  MoveL 5376 to (-21.97, 164.98, 78.65) mm, rotated rx 180 ry 0 rz 180 deg; joints [-137.804, 64.103, -73.918, 137.384, 82.745, 6.628]
  Call Extruder(394.83845)
  MoveL 5377 to (-22.56, 164.93, 78.65) mm, rotated rx -180 ry 0 rz 180 deg; joints [-137.905, 64.127, -73.891, 137.489, 82.771, 6.581]
  MoveL 5378 to (-22.56, 164.93, 78.65) mm, rotated rx -180 ry 0 rz 180 deg; joints [-137.905, 64.127, -73.891, 137.489, 82.771, 6.581]
  Call Extruder(395.13381)
  MoveL 5379 to (-23.15, 164.89, 78.65) mm, rotated rx 180 ry 0 rz -180 deg; joints [-138.004, 64.152, -73.865, 137.593, 82.796, 6.534]
  MoveL 5380 to (-23.15, 164.89, 78.65) mm, rotated rx 180 ry 0 rz -180 deg; joints [-138.004, 64.152, -73.865, 137.593, 82.796, 6.534]
  Call Extruder(395.38003)
  MoveL 5381 to (-23.64, 164.84, 78.65) mm, rotated rx 180 ry 0 rz 180 deg; joints [-138.088, 64.171, -73.843, 137.68, 82.818, 6.495]
  MoveL 5382 to (-23.64, 164.84, 78.65) mm, rotated rx 180 ry 0 rz 180 deg; joints [-138.088, 64.171, -73.843, 137.68, 82.818, 6.495]
  Call Extruder(395.57673)
  MoveL 5383 to (-24.03, 164.79, 78.65) mm, rotated rx 180 ry 0 rz 180 deg; joints [-138.156, 64.187, -73.827, 137.751, 82.834, 6.465]
  MoveL 5384 to (-24.03, 164.79, 78.65) mm, rotated rx 180 ry 0 rz 180 deg; joints [-138.156, 64.187, -73.827, 137.751, 82.834, 6.465]
  Call Extruder(395.77431)
  MoveL 5385 to (-24.42, 164.75, 78.65) mm, rotated rx 180 ry 0 rz 180 deg; joints [-138.224, 64.202, -73.81, 137.822, 82.85, 6.434]
  MoveL 5386 to (-24.42, 164.75, 78.65) mm, rotated rx 180 ry 0 rz 180 deg; joints [-138.224, 64.202, -73.81, 137.822, 82.85, 6.434]
  Call Extruder(395.97275)
  MoveL 5387 to (-24.8, 164.7, 78.65) mm, rotated rx -180 ry 0 rz -180 deg; joints [-138.292, 64.217, -73.793, 137.892, 82.866, 6.404]
  MoveL 5388 to (-24.8, 164.7, 78.65) mm, rotated rx -180 ry 0 rz -180 deg; joints [-138.292, 64.217, -73.793, 137.892, 82.866, 6.404]
  Call Extruder(396.17206)
  MoveL 5389 to (-25.19, 164.66, 78.65) mm, rotated rx 180 ry 0 rz 180 deg; joints [-138.359, 64.233, -73.776, 137.962, 82.883, 6.374]
  MoveL 5390 to (-25.19, 164.66, 78.65) mm, rotated rx 180 ry 0 rz 180 deg; joints [-138.359, 64.233, -73.776, 137.962, 82.883, 6.374]
  Call Extruder(396.33089)
  MoveL 5391 to (-25.5, 164.61, 78.65) mm, rotated rx -180 ry 0 rz 180 deg; joints [-138.415, 64.244, -73.763, 138.02, 82.895, 6.351]
  MoveL 5392 to (-25.5, 164.61, 78.65) mm, rotated rx -180 ry 0 rz 180 deg; joints [-138.415, 64.244, -73.763, 138.02, 82.895, 6.351]
  Call Extruder(396.49045)
  MoveL 5393 to (-25.8, 164.56, 78.65) mm, rotated rx -180 ry 0 rz 180 deg; joints [-138.47, 64.256, -73.75, 138.077, 82.907, 6.327]
  MoveL 5394 to (-25.8, 164.56, 78.65) mm, rotated rx -180 ry 0 rz 180 deg; joints [-138.47, 64.256, -73.75, 138.077, 82.907, 6.327]
  Call Extruder(396.65073)
  MoveL 5395 to (-26.11, 164.51, 78.65) mm, rotated rx 180 ry 0 rz 180 deg; joints [-138.525, 64.267, -73.737, 138.134, 82.919, 6.304]
  MoveL 5396 to (-26.11, 164.51, 78.65) mm, rotated rx 180 ry 0 rz 180 deg; joints [-138.525, 64.267, -73.737, 138.134, 82.919, 6.304]
  Call Extruder(396.81175)
  MoveL 5397 to (-26.41, 164.46, 78.65) mm, rotated rx 180 ry 0 rz 180 deg; joints [-138.58, 64.279, -73.724, 138.192, 82.931, 6.281]
  MoveL 5398 to (-26.41, 164.46, 78.65) mm, rotated rx 180 ry 0 rz 180 deg; joints [-138.58, 64.279, -73.724, 138.192, 82.931, 6.281]
  Call Extruder(396.97349)
  MoveL 5399 to (-26.72, 164.41, 78.65) mm, rotated rx 180 ry 0 rz 180 deg; joints [-138.635, 64.291, -73.711, 138.249, 82.944, 6.257]
  MoveL 5400 to (-26.72, 164.41, 78.65) mm, rotated rx 180 ry 0 rz 180 deg; joints [-138.635, 64.291, -73.711, 138.249, 82.944, 6.257]
  Call Extruder(397.13596)
  MoveL 5401 to (-27.03, 164.37, 78.65) mm, rotated rx 180 ry 0 rz 180 deg; joints [-138.69, 64.302, -73.698, 138.306, 82.956, 6.234]
  MoveL 5402 to (-27.03, 164.37, 78.65) mm, rotated rx 180 ry 0 rz 180 deg; joints [-138.69, 64.302, -73.698, 138.306, 82.956, 6.234]
  Call Extruder(397.26988)
  MoveL 5403 to (-27.27, 164.32, 78.65) mm, rotated rx -180 ry 0 rz 180 deg; joints [-138.736, 64.311, -73.688, 138.354, 82.965, 6.216]
  MoveL 5404 to (-27.27, 164.32, 78.65) mm, rotated rx -180 ry 0 rz 180 deg; joints [-138.736, 64.311, -73.688, 138.354, 82.965, 6.216]
  Call Extruder(397.40442)
  MoveL 5405 to (-27.52, 164.27, 78.65) mm, rotated rx 180 ry 0 rz 180 deg; joints [-138.783, 64.32, -73.678, 138.402, 82.975, 6.197]
  MoveL 5406 to (-27.52, 164.27, 78.65) mm, rotated rx 180 ry 0 rz 180 deg; joints [-138.783, 64.32, -73.678, 138.402, 82.975, 6.197]
  Call Extruder(397.53957)
  MoveL 5407 to (-27.77, 164.22, 78.65) mm, rotated rx 180 ry 0 rz 180 deg; joints [-138.829, 64.329, -73.668, 138.45, 82.984, 6.178]
  MoveL 5408 to (-27.77, 164.22, 78.65) mm, rotated rx 180 ry 0 rz 180 deg; joints [-138.829, 64.329, -73.668, 138.45, 82.984, 6.178]
  Call Extruder(397.67532)
  MoveL 5409 to (-28.02, 164.17, 78.65) mm, rotated rx -180 ry 0 rz 180 deg; joints [-138.875, 64.338, -73.657, 138.497, 82.994, 6.16]
  MoveL 5410 to (-28.02, 164.17, 78.65) mm, rotated rx -180 ry 0 rz 180 deg; joints [-138.875, 64.338, -73.657, 138.497, 82.994, 6.16]
  Call Extruder(397.81169)
  MoveL 5411 to (-28.27, 164.12, 78.65) mm, rotated rx -180 ry 0 rz -180 deg; joints [-138.921, 64.348, -73.647, 138.545, 83.003, 6.141]
  MoveL 5412 to (-28.27, 164.12, 78.65) mm, rotated rx -180 ry 0 rz -180 deg; joints [-138.921, 64.348, -73.647, 138.545, 83.003, 6.141]
  Call Extruder(397.89656)
  MoveL 5413 to (-28.42, 164.09, 78.65) mm, rotated rx -180 ry 0 rz 180 deg; joints [-138.95, 64.353, -73.641, 138.575, 83.009, 6.13]
  Set speed (130.0 mm/s)
  MoveL 5414 to (-31.76, 163.31, 78.65) mm, rotated rx -180 ry 0 rz 180 deg; joints [-139.581, 64.47, -73.506, 139.228, 83.133, 5.887]
  MoveL 5415 to (-31.76, 163.31, 88.06) mm, rotated rx -180 ry 0 rz -180 deg; joints [-139.581, 65.843, -75.425, 139.183, 82.719, 6.247]
  Call Extruder(395.89656)
  Set speed (40.0 mm/s)
  MoveL 5416 to (-31.76, 163.31, 88.06) mm, rotated rx -180 ry 0 rz -180 deg; joints [-139.581, 65.843, -75.425, 139.183, 82.719, 6.247]
  Call Extruder(0.00000)
  Set speed (130.0 mm/s)
  MoveL 5417 to (-31.64, 163.21, 88.06) mm, rotated rx -180 ry 0 rz 180 deg; joints [-139.581, 65.833, -75.436, 139.181, 82.704, 6.26]
  Call Extruder(2.00000)
  Set speed (40.0 mm/s)
  MoveL 5418 to (-31.64, 163.21, 88.06) mm, rotated rx -180 ry 0 rz 180 deg; joints [-139.581, 65.833, -75.436, 139.181, 82.704, 6.26]
  Set speed (30.0 mm/s)
  MoveL 5419 to (-31.64, 163.21, 88.06) mm, rotated rx -180 ry 0 rz 180 deg; joints [-139.581, 65.833, -75.436, 139.181, 82.704, 6.26]
  Call Extruder(2.18198)
  MoveL 5420 to (-31.93, 163.09, 88.06) mm, rotated rx -180 ry 0 rz 180 deg; joints [-139.645, 65.842, -75.426, 139.247, 82.711, 6.24]
  MoveL 5421 to (-31.93, 163.09, 88.06) mm, rotated rx -180 ry 0 rz 180 deg; joints [-139.645, 65.842, -75.426, 139.247, 82.711, 6.24]
  Call Extruder(2.36471)
  MoveL 5422 to (-32.22, 162.96, 88.06) mm, rotated rx -180 ry 0 rz 180 deg; joints [-139.709, 65.851, -75.416, 139.313, 82.718, 6.219]
  MoveL 5423 to (-32.22, 162.96, 88.06) mm, rotated rx -180 ry 0 rz 180 deg; joints [-139.709, 65.851, -75.416, 139.313, 82.718, 6.219]
  Call Extruder(2.53513)
  MoveL 5424 to (-32.49, 162.85, 88.06) mm, rotated rx -180 ry 0 rz -180 deg; joints [-139.768, 65.858, -75.407, 139.374, 82.724, 6.201]
  MoveL 5425 to (-32.49, 162.85, 88.06) mm, rotated rx -180 ry 0 rz -180 deg; joints [-139.768, 65.858, -75.407, 139.374, 82.724, 6.201]
  Call Extruder(2.69310)
  MoveL 5426 to (-32.74, 162.74, 88.06) mm, rotated rx -180 ry 0 rz 180 deg; joints [-139.823, 65.866, -75.399, 139.43, 82.73, 6.184]
  MoveL 5427 to (-32.74, 162.74, 88.06) mm, rotated rx -180 ry 0 rz 180 deg; joints [-139.823, 65.866, -75.399, 139.43, 82.73, 6.184]
  Call Extruder(2.85168)
  MoveL 5428 to (-32.99, 162.64, 88.06) mm, rotated rx -180 ry 0 rz 180 deg; joints [-139.878, 65.873, -75.391, 139.487, 82.736, 6.167]
  MoveL 5429 to (-32.99, 162.64, 88.06) mm, rotated rx -180 ry 0 rz 180 deg; joints [-139.878, 65.873, -75.391, 139.487, 82.736, 6.167]
  Call Extruder(3.05785)
  MoveL 5430 to (-33.29, 162.46, 88.06) mm, rotated rx -180 ry 0 rz 180 deg; joints [-139.953, 65.88, -75.383, 139.563, 82.739, 6.147]
  MoveL 5431 to (-33.29, 162.46, 88.06) mm, rotated rx -180 ry 0 rz 180 deg; joints [-139.953, 65.88, -75.383, 139.563, 82.739, 6.147]
  Call Extruder(3.26479)
  MoveL 5432 to (-33.6, 162.29, 88.06) mm, rotated rx -180 ry 0 rz 180 deg; joints [-140.028, 65.887, -75.375, 139.639, 82.743, 6.128]
  MoveL 5433 to (-33.6, 162.29, 88.06) mm, rotated rx -180 ry 0 rz 180 deg; joints [-140.028, 65.887, -75.375, 139.639, 82.743, 6.128]
  Call Extruder(3.47251)
  MoveL 5434 to (-33.9, 162.11, 88.06) mm, rotated rx 180 ry 0 rz -180 deg; joints [-140.103, 65.894, -75.367, 139.715, 82.746, 6.109]
  MoveL 5435 to (-33.9, 162.11, 88.06) mm, rotated rx 180 ry 0 rz -180 deg; joints [-140.103, 65.894, -75.367, 139.715, 82.746, 6.109]
  Call Extruder(3.68102)
  MoveL 5436 to (-34.21, 161.93, 88.06) mm, rotated rx -180 ry 0 rz 180 deg; joints [-140.178, 65.901, -75.359, 139.791, 82.75, 6.089]
  MoveL 5437 to (-34.21, 161.93, 88.06) mm, rotated rx -180 ry 0 rz 180 deg; joints [-140.178, 65.901, -75.359, 139.791, 82.75, 6.089]
  Call Extruder(3.86055)
  MoveL 5438 to (-34.45, 161.76, 88.06) mm, rotated rx -180 ry 0 rz 180 deg; joints [-140.244, 65.905, -75.354, 139.859, 82.75, 6.075]
  MoveL 5439 to (-34.45, 161.76, 88.06) mm, rotated rx -180 ry 0 rz 180 deg; joints [-140.244, 65.905, -75.354, 139.859, 82.75, 6.075]
  Call Extruder(4.19399)
  MoveL 5440 to (-34.9, 161.43, 88.06) mm, rotated rx 180 ry 0 rz 180 deg; joints [-140.366, 65.914, -75.344, 139.983, 82.75, 6.048]
  MoveL 5441 to (-34.9, 161.43, 88.06) mm, rotated rx 180 ry 0 rz 180 deg; joints [-140.366, 65.914, -75.344, 139.983, 82.75, 6.048]
  Call Extruder(4.52861)
  MoveL 5442 to (-35.35, 161.1, 88.06) mm, rotated rx -180 ry 0 rz -180 deg; joints [-140.489, 65.922, -75.335, 140.107, 82.751, 6.021]
  Call Extruder(5.35652)
  MoveL 5443 to (-36.39, 160.19, 88.06) mm, rotated rx -180 ry 0 rz -180 deg; joints [-140.797, 65.935, -75.32, 140.418, 82.741, 5.964]
  Call Extruder(6.18445)
  MoveL 5444 to (-37.3, 159.15, 88.06) mm, rotated rx 180 ry 0 rz 180 deg; joints [-141.109, 65.938, -75.316, 140.731, 82.714, 5.92]
  Call Extruder(6.35176)
  MoveL 5445 to (-37.47, 158.93, 88.06) mm, rotated rx 180 ry 0 rz 180 deg; joints [-141.172, 65.937, -75.317, 140.795, 82.706, 5.913]
  MoveL 5446 to (-37.47, 158.93, 88.06) mm, rotated rx 180 ry 0 rz 180 deg; joints [-141.172, 65.937, -75.317, 140.795, 82.706, 5.913]
  Call Extruder(6.68519)
  MoveL 5447 to (-37.79, 158.48, 88.06) mm, rotated rx -180 ry 0 rz 180 deg; joints [-141.298, 65.936, -75.319, 140.921, 82.69, 5.899]
  MoveL 5448 to (-37.79, 158.48, 88.06) mm, rotated rx -180 ry 0 rz 180 deg; joints [-141.298, 65.936, -75.319, 140.921, 82.69, 5.899]
  Call Extruder(7.01743)
  MoveL 5449 to (-38.12, 158.03, 88.06) mm, rotated rx -180 ry 0 rz 180 deg; joints [-141.424, 65.934, -75.321, 141.047, 82.675, 5.885]
  MoveL 5450 to (-38.12, 158.03, 88.06) mm, rotated rx -180 ry 0 rz 180 deg; joints [-141.424, 65.934, -75.321, 141.047, 82.675, 5.885]
  Call Extruder(7.13510)
  MoveL 5451 to (-38.22, 157.85, 88.06) mm, rotated rx 180 ry 0 rz -180 deg; joints [-141.468, 65.932, -75.323, 141.091, 82.667, 5.882]
  MoveL 5452 to (-38.22, 157.85, 88.06) mm, rotated rx 180 ry 0 rz -180 deg; joints [-141.468, 65.932, -75.323, 141.091, 82.667, 5.882]
  Call Extruder(7.34283)
  MoveL 5453 to (-38.4, 157.55, 88.06) mm, rotated rx -180 ry 0 rz 180 deg; joints [-141.547, 65.929, -75.326, 141.169, 82.654, 5.876]
  MoveL 5454 to (-38.4, 157.55, 88.06) mm, rotated rx -180 ry 0 rz 180 deg; joints [-141.547, 65.929, -75.326, 141.169, 82.654, 5.876]
  Call Extruder(7.54978)
  MoveL 5455 to (-38.57, 157.25, 88.06) mm, rotated rx -180 ry 0 rz 180 deg; joints [-141.625, 65.926, -75.329, 141.247, 82.641, 5.87]
  MoveL 5456 to (-38.57, 157.25, 88.06) mm, rotated rx -180 ry 0 rz 180 deg; joints [-141.625, 65.926, -75.329, 141.247, 82.641, 5.87]
  Call Extruder(7.75595)
  MoveL 5457 to (-38.75, 156.94, 88.06) mm, rotated rx 180 ry 0 rz 180 deg; joints [-141.704, 65.923, -75.333, 141.326, 82.628, 5.864]
  MoveL 5458 to (-38.75, 156.94, 88.06) mm, rotated rx 180 ry 0 rz 180 deg; joints [-141.704, 65.923, -75.333, 141.326, 82.628, 5.864]
  Call Extruder(7.93763)
  MoveL 5459 to (-38.89, 156.66, 88.06) mm, rotated rx -180 ry 0 rz 180 deg; joints [-141.773, 65.92, -75.337, 141.394, 82.615, 5.86]
  MoveL 5460 to (-38.89, 156.66, 88.06) mm, rotated rx -180 ry 0 rz 180 deg; joints [-141.773, 65.92, -75.337, 141.394, 82.615, 5.86]
  Call Extruder(8.09561)
  MoveL 5461 to (-39, 156.42, 88.06) mm, rotated rx -180 ry 0 rz 180 deg; joints [-141.832, 65.916, -75.342, 141.453, 82.602, 5.858]
  MoveL 5462 to (-39, 156.42, 88.06) mm, rotated rx -180 ry 0 rz 180 deg; joints [-141.832, 65.916, -75.342, 141.453, 82.602, 5.858]
  Call Extruder(8.25300)
  MoveL 5463 to (-39.11, 156.17, 88.06) mm, rotated rx -180 ry 0 rz 180 deg; joints [-141.891, 65.912, -75.346, 141.512, 82.589, 5.855]
  MoveL 5464 to (-39.11, 156.17, 88.06) mm, rotated rx -180 ry 0 rz 180 deg; joints [-141.891, 65.912, -75.346, 141.512, 82.589, 5.855]
  Call Extruder(8.43571)
  MoveL 5465 to (-39.23, 155.87, 88.06) mm, rotated rx -180 ry 0 rz -180 deg; joints [-141.96, 65.907, -75.352, 141.58, 82.574, 5.853]
  MoveL 5466 to (-39.23, 155.87, 88.06) mm, rotated rx -180 ry 0 rz -180 deg; joints [-141.96, 65.907, -75.352, 141.58, 82.574, 5.853]
  Call Extruder(8.61768)
  MoveL 5467 to (-39.35, 155.58, 88.06) mm, rotated rx 180 ry 0 rz 180 deg; joints [-142.029, 65.902, -75.358, 141.648, 82.558, 5.851]
  MoveL 5468 to (-39.35, 155.58, 88.06) mm, rotated rx 180 ry 0 rz 180 deg; joints [-142.029, 65.902, -75.358, 141.648, 82.558, 5.851]
  Call Extruder(8.76501)
  MoveL 5469 to (-39.44, 155.34, 88.06) mm, rotated rx 180 ry 0 rz -180 deg; joints [-142.085, 65.897, -75.363, 141.703, 82.545, 5.85]
  MoveL 5470 to (-39.44, 155.34, 88.06) mm, rotated rx 180 ry 0 rz -180 deg; joints [-142.085, 65.897, -75.363, 141.703, 82.545, 5.85]
  Call Extruder(8.87824)
  MoveL 5471 to (-39.5, 155.15, 88.06) mm, rotated rx -180 ry 0 rz -180 deg; joints [-142.127, 65.893, -75.367, 141.745, 82.534, 5.85]
  MoveL 5472 to (-39.5, 155.15, 88.06) mm, rotated rx -180 ry 0 rz -180 deg; joints [-142.127, 65.893, -75.367, 141.745, 82.534, 5.85]
  Call Extruder(8.99103)
  MoveL 5473 to (-39.56, 154.97, 88.06) mm, rotated rx 180 ry 0 rz 180 deg; joints [-142.169, 65.889, -75.372, 141.787, 82.523, 5.849]
  MoveL 5474 to (-39.56, 154.97, 88.06) mm, rotated rx 180 ry 0 rz 180 deg; joints [-142.169, 65.889, -75.372, 141.787, 82.523, 5.849]
  Call Extruder(9.10338)
  MoveL 5475 to (-39.62, 154.78, 88.06) mm, rotated rx -180 ry 0 rz 180 deg; joints [-142.212, 65.885, -75.377, 141.829, 82.512, 5.849]
  MoveL 5476 to (-39.62, 154.78, 88.06) mm, rotated rx -180 ry 0 rz 180 deg; joints [-142.212, 65.885, -75.377, 141.829, 82.512, 5.849]
  Call Extruder(9.21528)
  MoveL 5477 to (-39.68, 154.59, 88.06) mm, rotated rx -180 ry 0 rz -180 deg; joints [-142.254, 65.881, -75.381, 141.87, 82.501, 5.849]
  MoveL 5478 to (-39.68, 154.59, 88.06) mm, rotated rx -180 ry 0 rz -180 deg; joints [-142.254, 65.881, -75.381, 141.87, 82.501, 5.849]
  Call Extruder(9.33668)
  MoveL 5479 to (-39.75, 154.38, 88.06) mm, rotated rx -180 ry 0 rz 180 deg; joints [-142.3, 65.877, -75.386, 141.916, 82.489, 5.849]
  MoveL 5480 to (-39.75, 154.38, 88.06) mm, rotated rx -180 ry 0 rz 180 deg; joints [-142.3, 65.877, -75.386, 141.916, 82.489, 5.849]
  Call Extruder(9.46747)
  MoveL 5481 to (-39.82, 154.16, 88.06) mm, rotated rx 180 ry 0 rz 180 deg; joints [-142.35, 65.872, -75.392, 141.965, 82.476, 5.849]
  MoveL 5482 to (-39.82, 154.16, 88.06) mm, rotated rx 180 ry 0 rz 180 deg; joints [-142.35, 65.872, -75.392, 141.965, 82.476, 5.849]
  Call Extruder(9.59770)
  MoveL 5483 to (-39.88, 153.94, 88.06) mm, rotated rx 180 ry 0 rz -180 deg; joints [-142.399, 65.867, -75.397, 142.013, 82.463, 5.849]
  MoveL 5484 to (-39.88, 153.94, 88.06) mm, rotated rx 180 ry 0 rz -180 deg; joints [-142.399, 65.867, -75.397, 142.013, 82.463, 5.849]
  Call Extruder(9.72737)
  MoveL 5485 to (-39.95, 153.71, 88.06) mm, rotated rx -180 ry 0 rz -180 deg; joints [-142.449, 65.862, -75.403, 142.062, 82.449, 5.849]
  MoveL 5486 to (-39.95, 153.71, 88.06) mm, rotated rx -180 ry 0 rz -180 deg; joints [-142.449, 65.862, -75.403, 142.062, 82.449, 5.849]
  Call Extruder(9.85647)
  MoveL 5487 to (-40.02, 153.49, 88.06) mm, rotated rx -180 ry 0 rz 180 deg; joints [-142.498, 65.857, -75.408, 142.111, 82.436, 5.849]
  MoveL 5488 to (-40.02, 153.49, 88.06) mm, rotated rx -180 ry 0 rz 180 deg; joints [-142.498, 65.857, -75.408, 142.111, 82.436, 5.849]
  Call Extruder(9.97156)
  MoveL 5489 to (-40.06, 153.28, 88.06) mm, rotated rx -180 ry 0 rz 180 deg; joints [-142.541, 65.852, -75.414, 142.154, 82.423, 5.85]
  MoveL 5490 to (-40.06, 153.28, 88.06) mm, rotated rx -180 ry 0 rz 180 deg; joints [-142.541, 65.852, -75.414, 142.154, 82.423, 5.85]
  Call Extruder(10.08619)
  MoveL 5491 to (-40.11, 153.08, 88.06) mm, rotated rx 180 ry 0 rz 180 deg; joints [-142.584, 65.847, -75.42, 142.196, 82.41, 5.851]
  MoveL 5492 to (-40.11, 153.08, 88.06) mm, rotated rx 180 ry 0 rz 180 deg; joints [-142.584, 65.847, -75.42, 142.196, 82.41, 5.851]
  Call Extruder(10.20038)
  MoveL 5493 to (-40.15, 152.88, 88.06) mm, rotated rx 180 ry 0 rz 180 deg; joints [-142.627, 65.842, -75.426, 142.238, 82.396, 5.852]
  MoveL 5494 to (-40.15, 152.88, 88.06) mm, rotated rx 180 ry 0 rz 180 deg; joints [-142.627, 65.842, -75.426, 142.238, 82.396, 5.852]
  Call Extruder(10.31411)
  MoveL 5495 to (-40.2, 152.67, 88.06) mm, rotated rx -180 ry 0 rz 180 deg; joints [-142.671, 65.836, -75.432, 142.281, 82.383, 5.853]
  MoveL 5496 to (-40.2, 152.67, 88.06) mm, rotated rx -180 ry 0 rz 180 deg; joints [-142.671, 65.836, -75.432, 142.281, 82.383, 5.853]
  Call Extruder(10.43953)
  MoveL 5497 to (-40.24, 152.44, 88.06) mm, rotated rx 180 ry 0 rz 180 deg; joints [-142.718, 65.831, -75.439, 142.327, 82.368, 5.855]
  MoveL 5498 to (-40.24, 152.44, 88.06) mm, rotated rx 180 ry 0 rz 180 deg; joints [-142.718, 65.831, -75.439, 142.327, 82.368, 5.855]
  Call Extruder(10.57651)
  MoveL 5499 to (-40.29, 152.2, 88.06) mm, rotated rx 180 ry 0 rz 180 deg; joints [-142.77, 65.824, -75.446, 142.378, 82.352, 5.856]
  MoveL 5500 to (-40.29, 152.2, 88.06) mm, rotated rx 180 ry 0 rz 180 deg; joints [-142.77, 65.824, -75.446, 142.378, 82.352, 5.856]
  Call Extruder(10.71287)
  MoveL 5501 to (-40.34, 151.95, 88.06) mm, rotated rx -180 ry 0 rz 180 deg; joints [-142.822, 65.817, -75.454, 142.429, 82.335, 5.858]
  MoveL 5502 to (-40.34, 151.95, 88.06) mm, rotated rx -180 ry 0 rz 180 deg; joints [-142.822, 65.817, -75.454, 142.429, 82.335, 5.858]
  Call Extruder(10.84863)
  MoveL 5503 to (-40.39, 151.7, 88.06) mm, rotated rx 180 ry 0 rz 180 deg; joints [-142.874, 65.811, -75.461, 142.481, 82.319, 5.86]
  MoveL 5504 to (-40.39, 151.7, 88.06) mm, rotated rx 180 ry 0 rz 180 deg; joints [-142.874, 65.811, -75.461, 142.481, 82.319, 5.86]
  Call Extruder(10.98377)
  MoveL 5505 to (-40.44, 151.45, 88.06) mm, rotated rx -180 ry 0 rz 180 deg; joints [-142.926, 65.804, -75.468, 142.532, 82.303, 5.861]
  MoveL 5506 to (-40.44, 151.45, 88.06) mm, rotated rx -180 ry 0 rz 180 deg; joints [-142.926, 65.804, -75.468, 142.532, 82.303, 5.861]
  Call Extruder(11.11831)
  MoveL 5507 to (-40.49, 151.2, 88.06) mm, rotated rx 180 ry 0 rz 180 deg; joints [-142.978, 65.798, -75.476, 142.583, 82.286, 5.863]
  MoveL 5508 to (-40.49, 151.2, 88.06) mm, rotated rx 180 ry 0 rz 180 deg; joints [-142.978, 65.798, -75.476, 142.583, 82.286, 5.863]
  Call Extruder(11.25223)
  MoveL 5509 to (-40.54, 150.95, 88.06) mm, rotated rx 180 ry 0 rz 180 deg; joints [-143.031, 65.791, -75.483, 142.634, 82.27, 5.864]
  MoveL 5510 to (-40.54, 150.95, 88.06) mm, rotated rx 180 ry 0 rz 180 deg; joints [-143.031, 65.791, -75.483, 142.634, 82.27, 5.864]
  Call Extruder(11.40009)
  MoveL 5511 to (-40.59, 150.67, 88.06) mm, rotated rx 180 ry 0 rz 180 deg; joints [-143.088, 65.784, -75.492, 142.69, 82.251, 5.866]
  MoveL 5512 to (-40.59, 150.67, 88.06) mm, rotated rx 180 ry 0 rz 180 deg; joints [-143.088, 65.784, -75.492, 142.69, 82.251, 5.866]
  Call Extruder(11.56181)
  MoveL 5513 to (-40.64, 150.37, 88.06) mm, rotated rx -180 ry 0 rz 180 deg; joints [-143.15, 65.775, -75.501, 142.752, 82.23, 5.869]
  MoveL 5514 to (-40.64, 150.37, 88.06) mm, rotated rx -180 ry 0 rz 180 deg; joints [-143.15, 65.775, -75.501, 142.752, 82.23, 5.869]
  Call Extruder(11.72281)
  MoveL 5515 to (-40.69, 150.06, 88.06) mm, rotated rx -180 ry 0 rz 180 deg; joints [-143.213, 65.766, -75.511, 142.813, 82.209, 5.872]
  MoveL 5516 to (-40.69, 150.06, 88.06) mm, rotated rx -180 ry 0 rz 180 deg; joints [-143.213, 65.766, -75.511, 142.813, 82.209, 5.872]
  Call Extruder(11.88308)
  MoveL 5517 to (-40.74, 149.76, 88.06) mm, rotated rx -180 ry 0 rz 180 deg; joints [-143.276, 65.758, -75.52, 142.874, 82.189, 5.874]
  MoveL 5518 to (-40.74, 149.76, 88.06) mm, rotated rx -180 ry 0 rz 180 deg; joints [-143.276, 65.758, -75.52, 142.874, 82.189, 5.874]
  Call Extruder(12.04262)
  MoveL 5519 to (-40.78, 149.45, 88.06) mm, rotated rx -180 ry 0 rz -180 deg; joints [-143.338, 65.749, -75.53, 142.936, 82.168, 5.877]
  MoveL 5520 to (-40.78, 149.45, 88.06) mm, rotated rx -180 ry 0 rz -180 deg; joints [-143.338, 65.749, -75.53, 142.936, 82.168, 5.877]
  Call Extruder(12.20144)
  MoveL 5521 to (-40.83, 149.14, 88.06) mm, rotated rx 180 ry 0 rz 180 deg; joints [-143.401, 65.741, -75.54, 142.997, 82.147, 5.879]
  MoveL 5522 to (-40.83, 149.14, 88.06) mm, rotated rx 180 ry 0 rz 180 deg; joints [-143.401, 65.741, -75.54, 142.997, 82.147, 5.879]
  Call Extruder(12.38010)
  MoveL 5523 to (-40.88, 148.8, 88.06) mm, rotated rx -180 ry 0 rz 180 deg; joints [-143.471, 65.731, -75.551, 143.066, 82.123, 5.882]
  MoveL 5524 to (-40.88, 148.8, 88.06) mm, rotated rx -180 ry 0 rz 180 deg; joints [-143.471, 65.731, -75.551, 143.066, 82.123, 5.882]
  Call Extruder(12.57854)
  MoveL 5525 to (-40.92, 148.41, 88.06) mm, rotated rx -180 ry 0 rz 180 deg; joints [-143.549, 65.719, -75.564, 143.142, 82.095, 5.886]
  MoveL 5526 to (-40.92, 148.41, 88.06) mm, rotated rx -180 ry 0 rz 180 deg; joints [-143.549, 65.719, -75.564, 143.142, 82.095, 5.886]
  Call Extruder(12.77611)
  MoveL 5527 to (-40.97, 148.02, 88.06) mm, rotated rx -180 ry 0 rz -180 deg; joints [-143.627, 65.708, -75.576, 143.218, 82.068, 5.89]
  MoveL 5528 to (-40.97, 148.02, 88.06) mm, rotated rx -180 ry 0 rz -180 deg; joints [-143.627, 65.708, -75.576, 143.218, 82.068, 5.89]
  Call Extruder(12.97282)
  MoveL 5529 to (-41.02, 147.63, 88.06) mm, rotated rx -180 ry 0 rz -180 deg; joints [-143.705, 65.696, -75.589, 143.295, 82.04, 5.894]
  MoveL 5530 to (-41.02, 147.63, 88.06) mm, rotated rx -180 ry 0 rz -180 deg; joints [-143.705, 65.696, -75.589, 143.295, 82.04, 5.894]
  Call Extruder(13.16866)
  MoveL 5531 to (-41.06, 147.25, 88.06) mm, rotated rx -180 ry 0 rz 180 deg; joints [-143.783, 65.684, -75.602, 143.371, 82.013, 5.898]
  MoveL 5532 to (-41.06, 147.25, 88.06) mm, rotated rx -180 ry 0 rz 180 deg; joints [-143.783, 65.684, -75.602, 143.371, 82.013, 5.898]
  Call Extruder(13.46406)
  MoveL 5533 to (-41.11, 146.66, 88.06) mm, rotated rx -180 ry 0 rz -180 deg; joints [-143.899, 65.666, -75.622, 143.484, 81.97, 5.905]
  MoveL 5534 to (-41.11, 146.66, 88.06) mm, rotated rx -180 ry 0 rz -180 deg; joints [-143.899, 65.666, -75.622, 143.484, 81.97, 5.905]
  Call Extruder(13.75812)
  MoveL 5535 to (-41.16, 146.07, 88.06) mm, rotated rx -180 ry 0 rz 180 deg; joints [-144.015, 65.647, -75.643, 143.597, 81.926, 5.912]
  MoveL 5536 to (-41.16, 146.07, 88.06) mm, rotated rx -180 ry 0 rz 180 deg; joints [-144.015, 65.647, -75.643, 143.597, 81.926, 5.912]
  Call Extruder(14.05085)
  MoveL 5537 to (-41.2, 145.48, 88.06) mm, rotated rx -180 ry 0 rz 180 deg; joints [-144.131, 65.629, -75.663, 143.711, 81.883, 5.919]
  MoveL 5538 to (-41.2, 145.48, 88.06) mm, rotated rx -180 ry 0 rz 180 deg; joints [-144.131, 65.629, -75.663, 143.711, 81.883, 5.919]
  Call Extruder(14.62431)
  MoveL 5539 to (-41.25, 144.32, 88.06) mm, rotated rx -180 ry 0 rz -180 deg; joints [-144.355, 65.59, -75.705, 143.929, 81.795, 5.935]
  MoveL 5540 to (-41.25, 144.32, 88.06) mm, rotated rx -180 ry 0 rz -180 deg; joints [-144.355, 65.59, -75.705, 143.929, 81.795, 5.935]
  Call Extruder(15.33827)
  MoveL 5541 to (-41.29, 142.86, 88.06) mm, rotated rx 180 ry 0 rz 180 deg; joints [-144.635, 65.541, -75.758, 144.202, 81.683, 5.955]
  Call Extruder(57.40309)
  MoveL 5542 to (-41.29, 57.14, 88.06) mm, rotated rx -180 ry 0 rz -180 deg; joints [-164.153, 63.039, -77.935, 163.631, 75.682, 4.155]
  Call Extruder(57.83165)
  MoveL 5543 to (-41.27, 56.26, 88.06) mm, rotated rx -180 ry 0 rz 180 deg; joints [-164.382, 63.02, -77.948, 163.864, 75.636, 4.105]
  MoveL 5544 to (-41.27, 56.26, 88.06) mm, rotated rx -180 ry 0 rz 180 deg; joints [-164.382, 63.02, -77.948, 163.864, 75.636, 4.105]
  Call Extruder(58.40510)
  MoveL 5545 to (-41.23, 55.1, 88.06) mm, rotated rx -180 ry 0 rz 180 deg; joints [-164.686, 62.995, -77.965, 164.174, 75.572, 4.04]
  MoveL 5546 to (-41.23, 55.1, 88.06) mm, rotated rx -180 ry 0 rz 180 deg; joints [-164.686, 62.995, -77.965, 164.174, 75.572, 4.04]
  Call Extruder(58.83942)
  MoveL 5547 to (-41.18, 54.23, 88.06) mm, rotated rx -180 ry 0 rz 180 deg; joints [-164.915, 62.975, -77.979, 164.408, 75.524, 3.99]
  MoveL 5548 to (-41.18, 54.23, 88.06) mm, rotated rx -180 ry 0 rz 180 deg; joints [-164.915, 62.975, -77.979, 164.408, 75.524, 3.99]
  Call Extruder(59.13348)
  MoveL 5549 to (-41.13, 53.64, 88.06) mm, rotated rx 180 ry 0 rz 180 deg; joints [-165.068, 62.96, -77.989, 164.564, 75.49, 3.958]
  MoveL 5550 to (-41.13, 53.64, 88.06) mm, rotated rx 180 ry 0 rz 180 deg; joints [-165.068, 62.96, -77.989, 164.564, 75.49, 3.958]
  Call Extruder(59.42888)
  MoveL 5551 to (-41.09, 53.05, 88.06) mm, rotated rx -180 ry 0 rz 180 deg; joints [-165.222, 62.946, -77.999, 164.721, 75.456, 3.924]
  MoveL 5552 to (-41.09, 53.05, 88.06) mm, rotated rx -180 ry 0 rz 180 deg; joints [-165.222, 62.946, -77.999, 164.721, 75.456, 3.924]
  Call Extruder(59.67512)
  MoveL 5553 to (-41.04, 52.56, 88.06) mm, rotated rx -180 ry 0 rz -180 deg; joints [-165.349, 62.934, -78.008, 164.85, 75.427, 3.897]
  MoveL 5554 to (-41.04, 52.56, 88.06) mm, rotated rx -180 ry 0 rz -180 deg; joints [-165.349, 62.934, -78.008, 164.85, 75.427, 3.897]
  Call Extruder(59.87182)
  MoveL 5555 to (-40.99, 52.17, 88.06) mm, rotated rx 180 ry 0 rz 180 deg; joints [-165.449, 62.923, -78.015, 164.953, 75.404, 3.876]
  MoveL 5556 to (-40.99, 52.17, 88.06) mm, rotated rx 180 ry 0 rz 180 deg; joints [-165.449, 62.923, -78.015, 164.953, 75.404, 3.876]
  Call Extruder(60.06940)
  MoveL 5557 to (-40.95, 51.78, 88.06) mm, rotated rx -180 ry 0 rz 180 deg; joints [-165.549, 62.913, -78.022, 165.055, 75.38, 3.854]
  MoveL 5558 to (-40.95, 51.78, 88.06) mm, rotated rx -180 ry 0 rz 180 deg; joints [-165.549, 62.913, -78.022, 165.055, 75.38, 3.854]
  Call Extruder(60.26784)
  MoveL 5559 to (-40.9, 51.4, 88.06) mm, rotated rx -180 ry 0 rz -180 deg; joints [-165.65, 62.903, -78.029, 165.157, 75.357, 3.833]
  MoveL 5560 to (-40.9, 51.4, 88.06) mm, rotated rx -180 ry 0 rz -180 deg; joints [-165.65, 62.903, -78.029, 165.157, 75.357, 3.833]
  Call Extruder(60.46715)
  MoveL 5561 to (-40.86, 51.01, 88.06) mm, rotated rx -180 ry 0 rz -180 deg; joints [-165.751, 62.893, -78.036, 165.26, 75.333, 3.811]
  MoveL 5562 to (-40.86, 51.01, 88.06) mm, rotated rx -180 ry 0 rz -180 deg; joints [-165.751, 62.893, -78.036, 165.26, 75.333, 3.811]
  Call Extruder(60.62596)
  MoveL 5563 to (-40.81, 50.7, 88.06) mm, rotated rx 180 ry 0 rz 180 deg; joints [-165.829, 62.884, -78.042, 165.34, 75.314, 3.794]
  MoveL 5564 to (-40.81, 50.7, 88.06) mm, rotated rx 180 ry 0 rz 180 deg; joints [-165.829, 62.884, -78.042, 165.34, 75.314, 3.794]
  Call Extruder(60.78551)
  MoveL 5565 to (-40.76, 50.4, 88.06) mm, rotated rx 180 ry 0 rz -180 deg; joints [-165.908, 62.875, -78.048, 165.42, 75.294, 3.778]
  MoveL 5566 to (-40.76, 50.4, 88.06) mm, rotated rx 180 ry 0 rz -180 deg; joints [-165.908, 62.875, -78.048, 165.42, 75.294, 3.778]
  Call Extruder(60.94578)
  MoveL 5567 to (-40.71, 50.09, 88.06) mm, rotated rx -180 ry 0 rz 180 deg; joints [-165.987, 62.866, -78.054, 165.501, 75.274, 3.761]
  MoveL 5568 to (-40.71, 50.09, 88.06) mm, rotated rx -180 ry 0 rz 180 deg; joints [-165.987, 62.866, -78.054, 165.501, 75.274, 3.761]
  Call Extruder(61.10677)
  MoveL 5569 to (-40.66, 49.79, 88.06) mm, rotated rx -180 ry 0 rz -180 deg; joints [-166.066, 62.857, -78.06, 165.581, 75.255, 3.744]
  MoveL 5570 to (-40.66, 49.79, 88.06) mm, rotated rx -180 ry 0 rz -180 deg; joints [-166.066, 62.857, -78.06, 165.581, 75.255, 3.744]
  Call Extruder(61.26850)
  MoveL 5571 to (-40.61, 49.48, 88.06) mm, rotated rx -180 ry 0 rz 180 deg; joints [-166.145, 62.848, -78.066, 165.662, 75.235, 3.727]
  MoveL 5572 to (-40.61, 49.48, 88.06) mm, rotated rx -180 ry 0 rz 180 deg; joints [-166.145, 62.848, -78.066, 165.662, 75.235, 3.727]
  Call Extruder(61.43095)
  MoveL 5573 to (-40.57, 49.17, 88.06) mm, rotated rx 180 ry 0 rz -180 deg; joints [-166.224, 62.84, -78.072, 165.742, 75.216, 3.71]
  MoveL 5574 to (-40.57, 49.17, 88.06) mm, rotated rx 180 ry 0 rz -180 deg; joints [-166.224, 62.84, -78.072, 165.742, 75.216, 3.71]
  Call Extruder(61.56488)
  MoveL 5575 to (-40.52, 48.93, 88.06) mm, rotated rx 180 ry 0 rz -180 deg; joints [-166.288, 62.832, -78.078, 165.808, 75.199, 3.697]
  MoveL 5576 to (-40.52, 48.93, 88.06) mm, rotated rx 180 ry 0 rz -180 deg; joints [-166.288, 62.832, -78.078, 165.808, 75.199, 3.697]
  Call Extruder(61.69941)
  MoveL 5577 to (-40.47, 48.68, 88.06) mm, rotated rx -180 ry 0 rz 180 deg; joints [-166.352, 62.824, -78.083, 165.873, 75.182, 3.683]
  MoveL 5578 to (-40.47, 48.68, 88.06) mm, rotated rx -180 ry 0 rz 180 deg; joints [-166.352, 62.824, -78.083, 165.873, 75.182, 3.683]
  Call Extruder(61.83456)
  MoveL 5579 to (-40.42, 48.43, 88.06) mm, rotated rx 180 ry 0 rz 180 deg; joints [-166.416, 62.816, -78.088, 165.938, 75.165, 3.669]
  MoveL 5580 to (-40.42, 48.43, 88.06) mm, rotated rx 180 ry 0 rz 180 deg; joints [-166.416, 62.816, -78.088, 165.938, 75.165, 3.669]
  Call Extruder(61.97031)
  MoveL 5581 to (-40.37, 48.18, 88.06) mm, rotated rx -180 ry 0 rz 180 deg; joints [-166.48, 62.808, -78.093, 166.003, 75.148, 3.656]
  MoveL 5582 to (-40.37, 48.18, 88.06) mm, rotated rx -180 ry 0 rz 180 deg; joints [-166.48, 62.808, -78.093, 166.003, 75.148, 3.656]
  Call Extruder(62.10668)
  MoveL 5583 to (-40.32, 47.93, 88.06) mm, rotated rx 180 ry 0 rz 180 deg; joints [-166.544, 62.801, -78.099, 166.069, 75.132, 3.642]
  MoveL 5584 to (-40.32, 47.93, 88.06) mm, rotated rx 180 ry 0 rz 180 deg; joints [-166.544, 62.801, -78.099, 166.069, 75.132, 3.642]
  Call Extruder(62.24365)
  MoveL 5585 to (-40.27, 47.68, 88.06) mm, rotated rx -180 ry 0 rz -180 deg; joints [-166.608, 62.793, -78.104, 166.134, 75.115, 3.628]
  MoveL 5586 to (-40.27, 47.68, 88.06) mm, rotated rx -180 ry 0 rz -180 deg; joints [-166.608, 62.793, -78.104, 166.134, 75.115, 3.628]
  Call Extruder(62.38124)
  MoveL 5587 to (-40.22, 47.43, 88.06) mm, rotated rx -180 ry 0 rz -180 deg; joints [-166.673, 62.785, -78.109, 166.2, 75.098, 3.614]
  MoveL 5588 to (-40.22, 47.43, 88.06) mm, rotated rx -180 ry 0 rz -180 deg; joints [-166.673, 62.785, -78.109, 166.2, 75.098, 3.614]
  Call Extruder(62.49497)
  MoveL 5589 to (-40.17, 47.23, 88.06) mm, rotated rx -180 ry 0 rz -180 deg; joints [-166.725, 62.778, -78.114, 166.253, 75.084, 3.603]
  MoveL 5590 to (-40.17, 47.23, 88.06) mm, rotated rx -180 ry 0 rz -180 deg; joints [-166.725, 62.778, -78.114, 166.253, 75.084, 3.603]
  Call Extruder(62.60915)
  MoveL 5591 to (-40.13, 47.02, 88.06) mm, rotated rx -180 ry 0 rz 180 deg; joints [-166.778, 62.772, -78.118, 166.307, 75.07, 3.592]
  MoveL 5592 to (-40.13, 47.02, 88.06) mm, rotated rx -180 ry 0 rz 180 deg; joints [-166.778, 62.772, -78.118, 166.307, 75.07, 3.592]
  Call Extruder(62.72378)
  MoveL 5593 to (-40.08, 46.82, 88.06) mm, rotated rx -180 ry 0 rz -180 deg; joints [-166.83, 62.765, -78.123, 166.36, 75.056, 3.581]
  MoveL 5594 to (-40.08, 46.82, 88.06) mm, rotated rx -180 ry 0 rz -180 deg; joints [-166.83, 62.765, -78.123, 166.36, 75.056, 3.581]
  Call Extruder(62.83887)
  MoveL 5595 to (-40.04, 46.61, 88.06) mm, rotated rx -180 ry 0 rz -180 deg; joints [-166.883, 62.759, -78.127, 166.414, 75.042, 3.569]
  MoveL 5596 to (-40.04, 46.61, 88.06) mm, rotated rx -180 ry 0 rz -180 deg; joints [-166.883, 62.759, -78.127, 166.414, 75.042, 3.569]
  Call Extruder(62.96111)
  MoveL 5597 to (-39.98, 46.4, 88.06) mm, rotated rx -180 ry 0 rz -180 deg; joints [-166.937, 62.751, -78.132, 166.47, 75.026, 3.558]
  MoveL 5598 to (-39.98, 46.4, 88.06) mm, rotated rx -180 ry 0 rz -180 deg; joints [-166.937, 62.751, -78.132, 166.47, 75.026, 3.558]
  Call Extruder(63.09077)
  MoveL 5599 to (-39.92, 46.18, 88.06) mm, rotated rx 180 ry 0 rz 180 deg; joints [-166.994, 62.742, -78.138, 166.527, 75.009, 3.546]
  MoveL 5600 to (-39.92, 46.18, 88.06) mm, rotated rx 180 ry 0 rz 180 deg; joints [-166.994, 62.742, -78.138, 166.527, 75.009, 3.546]
  Call Extruder(63.22100)
  MoveL 5601 to (-39.85, 45.95, 88.06) mm, rotated rx 180 ry 0 rz 180 deg; joints [-167.051, 62.734, -78.144, 166.585, 74.992, 3.534]
  MoveL 5602 to (-39.85, 45.95, 88.06) mm, rotated rx 180 ry 0 rz 180 deg; joints [-167.051, 62.734, -78.144, 166.585, 74.992, 3.534]
  Call Extruder(63.35179)
  MoveL 5603 to (-39.78, 45.73, 88.06) mm, rotated rx 180 ry 0 rz -180 deg; joints [-167.107, 62.725, -78.149, 166.643, 74.974, 3.523]
  MoveL 5604 to (-39.78, 45.73, 88.06) mm, rotated rx 180 ry 0 rz -180 deg; joints [-167.107, 62.725, -78.149, 166.643, 74.974, 3.523]
  Call Extruder(63.48315)
  MoveL 5605 to (-39.71, 45.5, 88.06) mm, rotated rx -180 ry 0 rz 180 deg; joints [-167.164, 62.717, -78.155, 166.7, 74.957, 3.511]
  MoveL 5606 to (-39.71, 45.5, 88.06) mm, rotated rx -180 ry 0 rz 180 deg; joints [-167.164, 62.717, -78.155, 166.7, 74.957, 3.511]
  Call Extruder(63.59505)
  MoveL 5607 to (-39.65, 45.32, 88.06) mm, rotated rx -180 ry 0 rz 180 deg; joints [-167.212, 62.709, -78.16, 166.749, 74.942, 3.501]
  MoveL 5608 to (-39.65, 45.32, 88.06) mm, rotated rx -180 ry 0 rz 180 deg; joints [-167.212, 62.709, -78.16, 166.749, 74.942, 3.501]
  Call Extruder(63.70740)
  MoveL 5609 to (-39.59, 45.13, 88.06) mm, rotated rx -180 ry 0 rz -180 deg; joints [-167.26, 62.702, -78.165, 166.797, 74.927, 3.491]
  MoveL 5610 to (-39.59, 45.13, 88.06) mm, rotated rx -180 ry 0 rz -180 deg; joints [-167.26, 62.702, -78.165, 166.797, 74.927, 3.491]
  Call Extruder(63.82019)
  MoveL 5611 to (-39.53, 44.94, 88.06) mm, rotated rx -180 ry 0 rz -180 deg; joints [-167.307, 62.694, -78.17, 166.846, 74.912, 3.481]
  MoveL 5612 to (-39.53, 44.94, 88.06) mm, rotated rx -180 ry 0 rz -180 deg; joints [-167.307, 62.694, -78.17, 166.846, 74.912, 3.481]
  Call Extruder(63.93342)
  MoveL 5613 to (-39.47, 44.75, 88.06) mm, rotated rx 180 ry 0 rz -180 deg; joints [-167.355, 62.687, -78.175, 166.895, 74.897, 3.471]
  MoveL 5614 to (-39.47, 44.75, 88.06) mm, rotated rx 180 ry 0 rz -180 deg; joints [-167.355, 62.687, -78.175, 166.895, 74.897, 3.471]
  Call Extruder(64.04710)
  MoveL 5615 to (-39.41, 44.56, 88.06) mm, rotated rx 180 ry 0 rz -180 deg; joints [-167.403, 62.68, -78.18, 166.943, 74.882, 3.461]
  MoveL 5616 to (-39.41, 44.56, 88.06) mm, rotated rx 180 ry 0 rz -180 deg; joints [-167.403, 62.68, -78.18, 166.943, 74.882, 3.461]
  Call Extruder(64.22906)
  MoveL 5617 to (-39.29, 44.27, 88.06) mm, rotated rx 180 ry 0 rz 180 deg; joints [-167.475, 62.666, -78.189, 167.017, 74.856, 3.447]
  MoveL 5618 to (-39.29, 44.27, 88.06) mm, rotated rx 180 ry 0 rz 180 deg; joints [-167.475, 62.666, -78.189, 167.017, 74.856, 3.447]
  Call Extruder(64.41178)
  MoveL 5619 to (-39.17, 43.98, 88.06) mm, rotated rx -180 ry 0 rz -180 deg; joints [-167.548, 62.653, -78.198, 167.091, 74.83, 3.432]
  MoveL 5620 to (-39.17, 43.98, 88.06) mm, rotated rx -180 ry 0 rz -180 deg; joints [-167.548, 62.653, -78.198, 167.091, 74.83, 3.432]
  Call Extruder(64.58219)
  MoveL 5621 to (-39.05, 43.71, 88.06) mm, rotated rx 180 ry 0 rz 180 deg; joints [-167.615, 62.64, -78.206, 167.159, 74.806, 3.419]
  MoveL 5622 to (-39.05, 43.71, 88.06) mm, rotated rx 180 ry 0 rz 180 deg; joints [-167.615, 62.64, -78.206, 167.159, 74.806, 3.419]
  Call Extruder(64.74018)
  MoveL 5623 to (-38.94, 43.46, 88.06) mm, rotated rx -180 ry 0 rz -180 deg; joints [-167.677, 62.629, -78.213, 167.222, 74.783, 3.407]
  MoveL 5624 to (-38.94, 43.46, 88.06) mm, rotated rx -180 ry 0 rz -180 deg; joints [-167.677, 62.629, -78.213, 167.222, 74.783, 3.407]
  Call Extruder(64.89877)
  MoveL 5625 to (-38.84, 43.21, 88.06) mm, rotated rx -180 ry 0 rz 180 deg; joints [-167.739, 62.617, -78.221, 167.285, 74.76, 3.394]
  MoveL 5626 to (-38.84, 43.21, 88.06) mm, rotated rx -180 ry 0 rz 180 deg; joints [-167.739, 62.617, -78.221, 167.285, 74.76, 3.394]
  Call Extruder(65.10493)
  MoveL 5627 to (-38.66, 42.91, 88.06) mm, rotated rx -180 ry 0 rz -180 deg; joints [-167.813, 62.599, -78.233, 167.359, 74.728, 3.381]
  MoveL 5628 to (-38.66, 42.91, 88.06) mm, rotated rx -180 ry 0 rz -180 deg; joints [-167.813, 62.599, -78.233, 167.359, 74.728, 3.381]
  Call Extruder(65.31188)
  MoveL 5629 to (-38.49, 42.6, 88.06) mm, rotated rx 180 ry 0 rz 180 deg; joints [-167.886, 62.582, -78.244, 167.434, 74.695, 3.367]
  MoveL 5630 to (-38.49, 42.6, 88.06) mm, rotated rx 180 ry 0 rz 180 deg; joints [-167.886, 62.582, -78.244, 167.434, 74.695, 3.367]
  Call Extruder(65.51960)
  MoveL 5631 to (-38.31, 42.3, 88.06) mm, rotated rx -180 ry 0 rz -180 deg; joints [-167.96, 62.565, -78.255, 167.508, 74.663, 3.354]
  MoveL 5632 to (-38.31, 42.3, 88.06) mm, rotated rx -180 ry 0 rz -180 deg; joints [-167.96, 62.565, -78.255, 167.508, 74.663, 3.354]
  Call Extruder(65.72810)
  MoveL 5633 to (-38.13, 41.99, 88.06) mm, rotated rx -180 ry 0 rz -180 deg; joints [-168.033, 62.547, -78.267, 167.583, 74.63, 3.34]
  MoveL 5634 to (-38.13, 41.99, 88.06) mm, rotated rx -180 ry 0 rz -180 deg; joints [-168.033, 62.547, -78.267, 167.583, 74.63, 3.34]
  Call Extruder(65.90765)
  MoveL 5635 to (-37.96, 41.75, 88.06) mm, rotated rx -180 ry 0 rz -180 deg; joints [-168.091, 62.53, -78.277, 167.641, 74.6, 3.33]
  MoveL 5636 to (-37.96, 41.75, 88.06) mm, rotated rx -180 ry 0 rz -180 deg; joints [-168.091, 62.53, -78.277, 167.641, 74.6, 3.33]
  Call Extruder(66.24109)
  MoveL 5637 to (-37.63, 41.3, 88.06) mm, rotated rx 180 ry 0 rz -180 deg; joints [-168.197, 62.5, -78.297, 167.747, 74.545, 3.312]
  MoveL 5638 to (-37.63, 41.3, 88.06) mm, rotated rx 180 ry 0 rz -180 deg; joints [-168.197, 62.5, -78.297, 167.747, 74.545, 3.312]
  Call Extruder(66.57571)
  MoveL 5639 to (-37.3, 40.85, 88.06) mm, rotated rx -180 ry 0 rz -180 deg; joints [-168.304, 62.469, -78.317, 167.855, 74.489, 3.294]
  Call Extruder(67.40364)
  MoveL 5640 to (-36.39, 39.81, 88.06) mm, rotated rx -180 ry 0 rz 180 deg; joints [-168.541, 62.387, -78.37, 168.093, 74.344, 3.257]
  Call Extruder(68.23155)
  MoveL 5641 to (-35.35, 38.9, 88.06) mm, rotated rx 180 ry 0 rz -180 deg; joints [-168.739, 62.297, -78.426, 168.29, 74.189, 3.232]
  Call Extruder(68.39886)
  MoveL 5642 to (-35.13, 38.73, 88.06) mm, rotated rx 180 ry 0 rz 180 deg; joints [-168.773, 62.278, -78.438, 168.323, 74.157, 3.229]
  MoveL 5643 to (-35.13, 38.73, 88.06) mm, rotated rx 180 ry 0 rz 180 deg; joints [-168.773, 62.278, -78.438, 168.323, 74.157, 3.229]
  Call Extruder(68.73228)
  MoveL 5644 to (-34.68, 38.4, 88.06) mm, rotated rx 180 ry 0 rz 180 deg; joints [-168.84, 62.239, -78.462, 168.39, 74.093, 3.223]
  MoveL 5645 to (-34.68, 38.4, 88.06) mm, rotated rx 180 ry 0 rz 180 deg; joints [-168.84, 62.239, -78.462, 168.39, 74.093, 3.223]
  Call Extruder(69.06452)
  MoveL 5646 to (-34.23, 38.08, 88.06) mm, rotated rx -180 ry 0 rz 180 deg; joints [-168.908, 62.201, -78.485, 168.457, 74.028, 3.217]
  MoveL 5647 to (-34.23, 38.08, 88.06) mm, rotated rx -180 ry 0 rz 180 deg; joints [-168.908, 62.201, -78.485, 168.457, 74.028, 3.217]
  Call Extruder(69.18223)
  MoveL 5648 to (-34.05, 37.98, 88.06) mm, rotated rx -180 ry 0 rz -180 deg; joints [-168.927, 62.187, -78.494, 168.475, 74.005, 3.216]
  MoveL 5649 to (-34.05, 37.98, 88.06) mm, rotated rx -180 ry 0 rz -180 deg; joints [-168.927, 62.187, -78.494, 168.475, 74.005, 3.216]
  Call Extruder(69.38995)
  MoveL 5650 to (-33.75, 37.8, 88.06) mm, rotated rx -180 ry 0 rz -180 deg; joints [-168.96, 62.162, -78.509, 168.507, 73.963, 3.215]
  MoveL 5651 to (-33.75, 37.8, 88.06) mm, rotated rx -180 ry 0 rz -180 deg; joints [-168.96, 62.162, -78.509, 168.507, 73.963, 3.215]
  Call Extruder(69.59689)
  MoveL 5652 to (-33.45, 37.63, 88.06) mm, rotated rx -180 ry 0 rz 180 deg; joints [-168.993, 62.137, -78.525, 168.539, 73.921, 3.214]
  MoveL 5653 to (-33.45, 37.63, 88.06) mm, rotated rx -180 ry 0 rz 180 deg; joints [-168.993, 62.137, -78.525, 168.539, 73.921, 3.214]
  Call Extruder(69.80305)
  MoveL 5654 to (-33.14, 37.45, 88.06) mm, rotated rx -180 ry 0 rz -180 deg; joints [-169.026, 62.111, -78.54, 168.571, 73.88, 3.213]
  MoveL 5655 to (-33.14, 37.45, 88.06) mm, rotated rx -180 ry 0 rz -180 deg; joints [-169.026, 62.111, -78.54, 168.571, 73.88, 3.213]
  Call Extruder(69.98473)
  MoveL 5656 to (-32.87, 37.31, 88.06) mm, rotated rx -180 ry 0 rz 180 deg; joints [-169.052, 62.089, -78.554, 168.595, 73.843, 3.213]
  MoveL 5657 to (-32.87, 37.31, 88.06) mm, rotated rx -180 ry 0 rz 180 deg; joints [-169.052, 62.089, -78.554, 168.595, 73.843, 3.213]
  Call Extruder(70.14273)
  MoveL 5658 to (-32.62, 37.2, 88.06) mm, rotated rx -180 ry 0 rz -180 deg; joints [-169.068, 62.068, -78.566, 168.611, 73.81, 3.215]
  MoveL 5659 to (-32.62, 37.2, 88.06) mm, rotated rx -180 ry 0 rz -180 deg; joints [-169.068, 62.068, -78.566, 168.611, 73.81, 3.215]
  Call Extruder(70.30013)
  MoveL 5660 to (-32.37, 37.09, 88.06) mm, rotated rx -180 ry 0 rz -180 deg; joints [-169.085, 62.048, -78.578, 168.627, 73.777, 3.216]
  MoveL 5661 to (-32.37, 37.09, 88.06) mm, rotated rx -180 ry 0 rz -180 deg; joints [-169.085, 62.048, -78.578, 168.627, 73.777, 3.216]
  Call Extruder(70.48284)
  MoveL 5662 to (-32.08, 36.98, 88.06) mm, rotated rx 180 ry 0 rz 180 deg; joints [-169.104, 62.025, -78.592, 168.644, 73.739, 3.219]
  MoveL 5663 to (-32.08, 36.98, 88.06) mm, rotated rx 180 ry 0 rz 180 deg; joints [-169.104, 62.025, -78.592, 168.644, 73.739, 3.219]
  Call Extruder(70.66479)
  MoveL 5664 to (-31.78, 36.85, 88.06) mm, rotated rx 180 ry 0 rz 180 deg; joints [-169.122, 62.001, -78.606, 168.661, 73.701, 3.221]
  MoveL 5665 to (-31.78, 36.85, 88.06) mm, rotated rx 180 ry 0 rz 180 deg; joints [-169.122, 62.001, -78.606, 168.661, 73.701, 3.221]
  Call Extruder(70.81212)
  MoveL 5666 to (-31.54, 36.76, 88.06) mm, rotated rx 180 ry 0 rz 180 deg; joints [-169.135, 61.982, -78.618, 168.673, 73.67, 3.224]
  MoveL 5667 to (-31.54, 36.76, 88.06) mm, rotated rx 180 ry 0 rz 180 deg; joints [-169.135, 61.982, -78.618, 168.673, 73.67, 3.224]
  Call Extruder(70.92536)
  MoveL 5668 to (-31.35, 36.7, 88.06) mm, rotated rx 180 ry 0 rz 180 deg; joints [-169.143, 61.967, -78.627, 168.679, 73.646, 3.226]
  MoveL 5669 to (-31.35, 36.7, 88.06) mm, rotated rx 180 ry 0 rz 180 deg; joints [-169.143, 61.967, -78.627, 168.679, 73.646, 3.226]
  Call Extruder(71.03815)
  MoveL 5670 to (-31.17, 36.64, 88.06) mm, rotated rx 180 ry 0 rz 180 deg; joints [-169.15, 61.952, -78.636, 168.685, 73.623, 3.229]
  MoveL 5671 to (-31.17, 36.64, 88.06) mm, rotated rx 180 ry 0 rz 180 deg; joints [-169.15, 61.952, -78.636, 168.685, 73.623, 3.229]
  Call Extruder(71.15050)
  MoveL 5672 to (-30.98, 36.58, 88.06) mm, rotated rx -180 ry 0 rz 180 deg; joints [-169.157, 61.936, -78.645, 168.691, 73.599, 3.232]
  MoveL 5673 to (-30.98, 36.58, 88.06) mm, rotated rx -180 ry 0 rz 180 deg; joints [-169.157, 61.936, -78.645, 168.691, 73.599, 3.232]
  Call Extruder(71.26240)
  MoveL 5674 to (-30.79, 36.52, 88.06) mm, rotated rx 180 ry 0 rz 180 deg; joints [-169.164, 61.921, -78.654, 168.697, 73.575, 3.235]
  MoveL 5675 to (-30.79, 36.52, 88.06) mm, rotated rx 180 ry 0 rz 180 deg; joints [-169.164, 61.921, -78.654, 168.697, 73.575, 3.235]
  Call Extruder(71.38380)
  MoveL 5676 to (-30.58, 36.45, 88.06) mm, rotated rx -180 ry 0 rz 180 deg; joints [-169.172, 61.905, -78.663, 168.704, 73.549, 3.238]
  MoveL 5677 to (-30.58, 36.45, 88.06) mm, rotated rx -180 ry 0 rz 180 deg; joints [-169.172, 61.905, -78.663, 168.704, 73.549, 3.238]
  Call Extruder(71.51459)
  MoveL 5678 to (-30.36, 36.39, 88.06) mm, rotated rx -180 ry 0 rz -180 deg; joints [-169.179, 61.887, -78.674, 168.71, 73.52, 3.241]
  MoveL 5679 to (-30.36, 36.39, 88.06) mm, rotated rx -180 ry 0 rz -180 deg; joints [-169.179, 61.887, -78.674, 168.71, 73.52, 3.241]
  Call Extruder(71.64482)
  MoveL 5680 to (-30.14, 36.32, 88.06) mm, rotated rx -180 ry 0 rz -180 deg; joints [-169.186, 61.869, -78.684, 168.715, 73.492, 3.245]
  MoveL 5681 to (-30.14, 36.32, 88.06) mm, rotated rx -180 ry 0 rz -180 deg; joints [-169.186, 61.869, -78.684, 168.715, 73.492, 3.245]
  Call Extruder(71.77448)
  MoveL 5682 to (-29.91, 36.25, 88.06) mm, rotated rx -180 ry 0 rz 180 deg; joints [-169.193, 61.851, -78.695, 168.721, 73.464, 3.249]
  MoveL 5683 to (-29.91, 36.25, 88.06) mm, rotated rx -180 ry 0 rz 180 deg; joints [-169.193, 61.851, -78.695, 168.721, 73.464, 3.249]
  Call Extruder(71.90358)
  MoveL 5684 to (-29.69, 36.18, 88.06) mm, rotated rx -180 ry 0 rz -180 deg; joints [-169.201, 61.833, -78.705, 168.727, 73.436, 3.252]
  MoveL 5685 to (-29.69, 36.18, 88.06) mm, rotated rx -180 ry 0 rz -180 deg; joints [-169.201, 61.833, -78.705, 168.727, 73.436, 3.252]
  Call Extruder(72.01865)
  MoveL 5686 to (-29.48, 36.14, 88.06) mm, rotated rx -180 ry 0 rz 180 deg; joints [-169.202, 61.817, -78.714, 168.727, 73.411, 3.257]
  MoveL 5687 to (-29.48, 36.14, 88.06) mm, rotated rx -180 ry 0 rz 180 deg; joints [-169.202, 61.817, -78.714, 168.727, 73.411, 3.257]
  Call Extruder(72.13327)
  MoveL 5688 to (-29.28, 36.09, 88.06) mm, rotated rx -180 ry 0 rz -180 deg; joints [-169.204, 61.801, -78.724, 168.728, 73.386, 3.262]
  MoveL 5689 to (-29.28, 36.09, 88.06) mm, rotated rx -180 ry 0 rz -180 deg; joints [-169.204, 61.801, -78.724, 168.728, 73.386, 3.262]
  Call Extruder(72.24744)
  MoveL 5690 to (-29.08, 36.05, 88.06) mm, rotated rx -180 ry 0 rz 180 deg; joints [-169.206, 61.785, -78.733, 168.728, 73.361, 3.266]
  MoveL 5691 to (-29.08, 36.05, 88.06) mm, rotated rx -180 ry 0 rz 180 deg; joints [-169.206, 61.785, -78.733, 168.728, 73.361, 3.266]
  Call Extruder(72.36115)
  MoveL 5692 to (-28.87, 36, 88.06) mm, rotated rx -180 ry 0 rz 180 deg; joints [-169.207, 61.769, -78.742, 168.728, 73.336, 3.271]
  MoveL 5693 to (-28.87, 36, 88.06) mm, rotated rx -180 ry 0 rz 180 deg; joints [-169.207, 61.769, -78.742, 168.728, 73.336, 3.271]
  Call Extruder(72.48657)
  MoveL 5694 to (-28.64, 35.96, 88.06) mm, rotated rx 180 ry 0 rz 180 deg; joints [-169.208, 61.751, -78.752, 168.728, 73.308, 3.277]
  MoveL 5695 to (-28.64, 35.96, 88.06) mm, rotated rx 180 ry 0 rz 180 deg; joints [-169.208, 61.751, -78.752, 168.728, 73.308, 3.277]
  Call Extruder(72.62355)
  MoveL 5696 to (-28.4, 35.91, 88.06) mm, rotated rx -180 ry 0 rz 180 deg; joints [-169.209, 61.731, -78.764, 168.727, 73.278, 3.283]
  MoveL 5697 to (-28.4, 35.91, 88.06) mm, rotated rx -180 ry 0 rz 180 deg; joints [-169.209, 61.731, -78.764, 168.727, 73.278, 3.283]
  Call Extruder(72.75992)
  MoveL 5698 to (-28.15, 35.86, 88.06) mm, rotated rx 180 ry 0 rz 180 deg; joints [-169.21, 61.712, -78.775, 168.725, 73.247, 3.289]
  MoveL 5699 to (-28.15, 35.86, 88.06) mm, rotated rx 180 ry 0 rz 180 deg; joints [-169.21, 61.712, -78.775, 168.725, 73.247, 3.289]
  Call Extruder(72.89567)
  MoveL 5700 to (-27.9, 35.81, 88.06) mm, rotated rx -180 ry 0 rz 180 deg; joints [-169.21, 61.692, -78.786, 168.724, 73.217, 3.295]
  MoveL 5701 to (-27.9, 35.81, 88.06) mm, rotated rx -180 ry 0 rz 180 deg; joints [-169.21, 61.692, -78.786, 168.724, 73.217, 3.295]
  Call Extruder(73.03082)
  MoveL 5702 to (-27.65, 35.76, 88.06) mm, rotated rx -180 ry 0 rz -180 deg; joints [-169.211, 61.672, -78.797, 168.723, 73.187, 3.301]
  MoveL 5703 to (-27.65, 35.76, 88.06) mm, rotated rx -180 ry 0 rz -180 deg; joints [-169.211, 61.672, -78.797, 168.723, 73.187, 3.301]
  Call Extruder(73.16536)
  MoveL 5704 to (-27.4, 35.71, 88.06) mm, rotated rx -180 ry 0 rz -180 deg; joints [-169.212, 61.652, -78.808, 168.722, 73.156, 3.307]
  MoveL 5705 to (-27.4, 35.71, 88.06) mm, rotated rx -180 ry 0 rz -180 deg; joints [-169.212, 61.652, -78.808, 168.722, 73.156, 3.307]
  Call Extruder(73.29928)
  MoveL 5706 to (-27.15, 35.66, 88.06) mm, rotated rx -180 ry 0 rz -180 deg; joints [-169.212, 61.633, -78.819, 168.72, 73.126, 3.313]
  MoveL 5707 to (-27.15, 35.66, 88.06) mm, rotated rx -180 ry 0 rz -180 deg; joints [-169.212, 61.633, -78.819, 168.72, 73.126, 3.313]
  Call Extruder(73.44714)
  MoveL 5708 to (-26.87, 35.61, 88.06) mm, rotated rx 180 ry 0 rz 180 deg; joints [-169.211, 61.611, -78.832, 168.717, 73.093, 3.321]
  MoveL 5709 to (-26.87, 35.61, 88.06) mm, rotated rx 180 ry 0 rz 180 deg; joints [-169.211, 61.611, -78.832, 168.717, 73.093, 3.321]
  Call Extruder(73.60888)
  MoveL 5710 to (-26.57, 35.56, 88.06) mm, rotated rx -180 ry 0 rz -180 deg; joints [-169.208, 61.587, -78.845, 168.712, 73.056, 3.329]
  MoveL 5711 to (-26.57, 35.56, 88.06) mm, rotated rx -180 ry 0 rz -180 deg; joints [-169.208, 61.587, -78.845, 168.712, 73.056, 3.329]
  Call Extruder(73.76989)
  MoveL 5712 to (-26.26, 35.51, 88.06) mm, rotated rx 180 ry 0 rz -180 deg; joints [-169.205, 61.562, -78.859, 168.707, 73.019, 3.338]
  MoveL 5713 to (-26.26, 35.51, 88.06) mm, rotated rx 180 ry 0 rz -180 deg; joints [-169.205, 61.562, -78.859, 168.707, 73.019, 3.338]
  Call Extruder(73.93017)
  MoveL 5714 to (-25.96, 35.47, 88.06) mm, rotated rx 180 ry 0 rz -180 deg; joints [-169.202, 61.538, -78.872, 168.702, 72.983, 3.346]
  MoveL 5715 to (-25.96, 35.47, 88.06) mm, rotated rx 180 ry 0 rz -180 deg; joints [-169.202, 61.538, -78.872, 168.702, 72.983, 3.346]
  Call Extruder(74.08972)
  MoveL 5716 to (-25.65, 35.42, 88.06) mm, rotated rx 180 ry 0 rz 180 deg; joints [-169.199, 61.514, -78.885, 168.696, 72.946, 3.355]
  MoveL 5717 to (-25.65, 35.42, 88.06) mm, rotated rx 180 ry 0 rz 180 deg; joints [-169.199, 61.514, -78.885, 168.696, 72.946, 3.355]
  Call Extruder(74.24855)
  MoveL 5718 to (-25.34, 35.37, 88.06) mm, rotated rx 180 ry 0 rz 180 deg; joints [-169.196, 61.49, -78.899, 168.691, 72.909, 3.364]
  MoveL 5719 to (-25.34, 35.37, 88.06) mm, rotated rx 180 ry 0 rz 180 deg; joints [-169.196, 61.49, -78.899, 168.691, 72.909, 3.364]
  Call Extruder(74.42721)
  MoveL 5720 to (-25, 35.32, 88.06) mm, rotated rx -180 ry 0 rz -180 deg; joints [-169.191, 61.463, -78.914, 168.682, 72.868, 3.374]
  MoveL 5721 to (-25, 35.32, 88.06) mm, rotated rx -180 ry 0 rz -180 deg; joints [-169.191, 61.463, -78.914, 168.682, 72.868, 3.374]
  Call Extruder(74.62566)
  MoveL 5722 to (-24.61, 35.27, 88.06) mm, rotated rx -180 ry 0 rz 180 deg; joints [-169.182, 61.432, -78.93, 168.671, 72.822, 3.386]
  MoveL 5723 to (-24.61, 35.27, 88.06) mm, rotated rx -180 ry 0 rz 180 deg; joints [-169.182, 61.432, -78.93, 168.671, 72.822, 3.386]
  Call Extruder(74.82323)
  MoveL 5724 to (-24.22, 35.23, 88.06) mm, rotated rx 180 ry 0 rz 180 deg; joints [-169.174, 61.401, -78.947, 168.659, 72.776, 3.399]
  MoveL 5725 to (-24.22, 35.23, 88.06) mm, rotated rx 180 ry 0 rz 180 deg; joints [-169.174, 61.401, -78.947, 168.659, 72.776, 3.399]
  Call Extruder(75.01994)
  MoveL 5726 to (-23.83, 35.18, 88.06) mm, rotated rx 180 ry 0 rz 180 deg; joints [-169.166, 61.371, -78.964, 168.647, 72.731, 3.411]
  MoveL 5727 to (-23.83, 35.18, 88.06) mm, rotated rx 180 ry 0 rz 180 deg; joints [-169.166, 61.371, -78.964, 168.647, 72.731, 3.411]
  Call Extruder(75.21578)
  MoveL 5728 to (-23.45, 35.14, 88.06) mm, rotated rx -180 ry 0 rz -180 deg; joints [-169.157, 61.34, -78.98, 168.635, 72.685, 3.423]
  MoveL 5729 to (-23.45, 35.14, 88.06) mm, rotated rx -180 ry 0 rz -180 deg; joints [-169.157, 61.34, -78.98, 168.635, 72.685, 3.423]
  Call Extruder(75.51117)
  MoveL 5730 to (-22.86, 35.09, 88.06) mm, rotated rx -180 ry 0 rz -180 deg; joints [-169.137, 61.294, -79.005, 168.61, 72.616, 3.444]
  MoveL 5731 to (-22.86, 35.09, 88.06) mm, rotated rx -180 ry 0 rz -180 deg; joints [-169.137, 61.294, -79.005, 168.61, 72.616, 3.444]
  Call Extruder(75.80523)
  MoveL 5732 to (-22.27, 35.04, 88.06) mm, rotated rx -180 ry 0 rz -180 deg; joints [-169.117, 61.247, -79.03, 168.584, 72.548, 3.465]
  MoveL 5733 to (-22.27, 35.04, 88.06) mm, rotated rx -180 ry 0 rz -180 deg; joints [-169.117, 61.247, -79.03, 168.584, 72.548, 3.465]
  Call Extruder(76.09796)
  MoveL 5734 to (-21.68, 35, 88.06) mm, rotated rx -180 ry 0 rz 180 deg; joints [-169.096, 61.2, -79.054, 168.559, 72.479, 3.487]
  MoveL 5735 to (-21.68, 35, 88.06) mm, rotated rx -180 ry 0 rz 180 deg; joints [-169.096, 61.2, -79.054, 168.559, 72.479, 3.487]
  Call Extruder(76.67141)
  MoveL 5736 to (-20.52, 34.95, 88.06) mm, rotated rx 180 ry 0 rz 180 deg; joints [-169.042, 61.109, -79.102, 168.493, 72.346, 3.533]
  MoveL 5737 to (-20.52, 34.95, 88.06) mm, rotated rx 180 ry 0 rz 180 deg; joints [-169.042, 61.109, -79.102, 168.493, 72.346, 3.533]
  Call Extruder(77.38537)
  MoveL 5738 to (-19.06, 34.91, 88.06) mm, rotated rx 180 ry 0 rz 180 deg; joints [-168.967, 60.994, -79.161, 168.404, 72.181, 3.593]
  Call Extruder(194.23211)
  MoveL 5739 to (219.06, 34.91, 88.06) mm, rotated rx 180 ry 0 rz 180 deg; joints [-30.588, 50.162, -81.339, 34.64, 116.465, 17.113]
  Call Extruder(194.66067)
  MoveL 5740 to (219.94, 34.93, 88.06) mm, rotated rx -180 ry 0 rz 180 deg; joints [-30.233, 50.245, -81.341, 34.239, 116.501, 16.893]
  MoveL 5741 to (219.94, 34.93, 88.06) mm, rotated rx -180 ry 0 rz 180 deg; joints [-30.233, 50.245, -81.341, 34.239, 116.501, 16.893]
  Call Extruder(195.23412)
  MoveL 5742 to (221.1, 34.98, 88.06) mm, rotated rx 180 ry 0 rz 180 deg; joints [-29.789, 50.357, -81.343, 33.732, 116.539, 16.612]
  MoveL 5743 to (221.1, 34.98, 88.06) mm, rotated rx 180 ry 0 rz 180 deg; joints [-29.789, 50.357, -81.343, 33.732, 116.539, 16.612]
  Call Extruder(195.66843)
  MoveL 5744 to (221.97, 35.02, 88.06) mm, rotated rx 180 ry 0 rz 180 deg; joints [-29.47, 50.442, -81.344, 33.368, 116.559, 16.408]
  MoveL 5745 to (221.97, 35.02, 88.06) mm, rotated rx 180 ry 0 rz 180 deg; joints [-29.47, 50.442, -81.344, 33.368, 116.559, 16.408]
  Call Extruder(195.96249)
  MoveL 5746 to (222.56, 35.07, 88.06) mm, rotated rx 180 ry 0 rz 180 deg; joints [-29.272, 50.5, -81.345, 33.139, 116.567, 16.277]
  MoveL 5747 to (222.56, 35.07, 88.06) mm, rotated rx 180 ry 0 rz 180 deg; joints [-29.272, 50.5, -81.345, 33.139, 116.567, 16.277]
  Call Extruder(196.25788)
  MoveL 5748 to (223.15, 35.11, 88.06) mm, rotated rx -180 ry 0 rz 180 deg; joints [-29.075, 50.558, -81.345, 32.912, 116.574, 16.148]
  MoveL 5749 to (223.15, 35.11, 88.06) mm, rotated rx -180 ry 0 rz 180 deg; joints [-29.075, 50.558, -81.345, 32.912, 116.574, 16.148]
  Call Extruder(196.50411)
  MoveL 5750 to (223.64, 35.16, 88.06) mm, rotated rx -180 ry 0 rz 180 deg; joints [-28.92, 50.606, -81.346, 32.732, 116.577, 16.044]
  MoveL 5751 to (223.64, 35.16, 88.06) mm, rotated rx -180 ry 0 rz 180 deg; joints [-28.92, 50.606, -81.346, 32.732, 116.577, 16.044]
  Call Extruder(196.70082)
  MoveL 5752 to (224.03, 35.21, 88.06) mm, rotated rx 180 ry 0 rz 180 deg; joints [-28.804, 50.645, -81.346, 32.598, 116.576, 15.965]
  MoveL 5753 to (224.03, 35.21, 88.06) mm, rotated rx 180 ry 0 rz 180 deg; joints [-28.804, 50.645, -81.346, 32.598, 116.576, 15.965]
  Call Extruder(196.89840)
  MoveL 5754 to (224.42, 35.25, 88.06) mm, rotated rx -180 ry 0 rz 180 deg; joints [-28.69, 50.684, -81.346, 32.465, 116.575, 15.887]
  MoveL 5755 to (224.42, 35.25, 88.06) mm, rotated rx -180 ry 0 rz 180 deg; joints [-28.69, 50.684, -81.346, 32.465, 116.575, 15.887]
  Call Extruder(197.09684)
  MoveL 5756 to (224.8, 35.3, 88.06) mm, rotated rx -180 ry 0 rz 180 deg; joints [-28.577, 50.723, -81.347, 32.332, 116.573, 15.809]
  MoveL 5757 to (224.8, 35.3, 88.06) mm, rotated rx -180 ry 0 rz 180 deg; joints [-28.577, 50.723, -81.347, 32.332, 116.573, 15.809]
  Call Extruder(197.29615)
  MoveL 5758 to (225.19, 35.34, 88.06) mm, rotated rx 180 ry 0 rz 180 deg; joints [-28.465, 50.762, -81.347, 32.202, 116.57, 15.732]
  MoveL 5759 to (225.19, 35.34, 88.06) mm, rotated rx 180 ry 0 rz 180 deg; joints [-28.465, 50.762, -81.347, 32.202, 116.57, 15.732]
  Call Extruder(197.45497)
  MoveL 5760 to (225.5, 35.39, 88.06) mm, rotated rx -180 ry 0 rz 180 deg; joints [-28.385, 50.794, -81.347, 32.108, 116.566, 15.675]
  MoveL 5761 to (225.5, 35.39, 88.06) mm, rotated rx -180 ry 0 rz 180 deg; joints [-28.385, 50.794, -81.347, 32.108, 116.566, 15.675]
  Call Extruder(197.61452)
  MoveL 5762 to (225.8, 35.44, 88.06) mm, rotated rx 180 ry 0 rz -180 deg; joints [-28.307, 50.825, -81.347, 32.015, 116.56, 15.619]
  MoveL 5763 to (225.8, 35.44, 88.06) mm, rotated rx 180 ry 0 rz -180 deg; joints [-28.307, 50.825, -81.347, 32.015, 116.56, 15.619]
  Call Extruder(197.77480)
  MoveL 5764 to (226.11, 35.49, 88.06) mm, rotated rx 180 ry 0 rz 180 deg; joints [-28.228, 50.856, -81.347, 31.922, 116.555, 15.563]
  MoveL 5765 to (226.11, 35.49, 88.06) mm, rotated rx 180 ry 0 rz 180 deg; joints [-28.228, 50.856, -81.347, 31.922, 116.555, 15.563]
  Call Extruder(197.93580)
  MoveL 5766 to (226.41, 35.54, 88.06) mm, rotated rx -180 ry 0 rz 180 deg; joints [-28.151, 50.888, -81.347, 31.831, 116.549, 15.507]
  MoveL 5767 to (226.41, 35.54, 88.06) mm, rotated rx -180 ry 0 rz 180 deg; joints [-28.151, 50.888, -81.347, 31.831, 116.549, 15.507]
  Call Extruder(198.09753)
  MoveL 5768 to (226.72, 35.59, 88.06) mm, rotated rx -180 ry 0 rz -180 deg; joints [-28.074, 50.919, -81.347, 31.739, 116.543, 15.451]
  MoveL 5769 to (226.72, 35.59, 88.06) mm, rotated rx -180 ry 0 rz -180 deg; joints [-28.074, 50.919, -81.347, 31.739, 116.543, 15.451]
  Call Extruder(198.25999)
  MoveL 5770 to (227.02, 35.63, 88.06) mm, rotated rx -180 ry 0 rz 180 deg; joints [-27.998, 50.95, -81.347, 31.649, 116.536, 15.396]
  MoveL 5771 to (227.02, 35.63, 88.06) mm, rotated rx -180 ry 0 rz 180 deg; joints [-27.998, 50.95, -81.347, 31.649, 116.536, 15.396]
  Call Extruder(198.39392)
  MoveL 5772 to (227.28, 35.68, 88.06) mm, rotated rx -180 ry 0 rz -180 deg; joints [-27.942, 50.976, -81.347, 31.582, 116.528, 15.354]
  MoveL 5773 to (227.28, 35.68, 88.06) mm, rotated rx -180 ry 0 rz -180 deg; joints [-27.942, 50.976, -81.347, 31.582, 116.528, 15.354]
  Call Extruder(198.52846)
  MoveL 5774 to (227.52, 35.73, 88.06) mm, rotated rx -180 ry 0 rz 180 deg; joints [-27.888, 51.003, -81.346, 31.517, 116.52, 15.313]
  MoveL 5775 to (227.52, 35.73, 88.06) mm, rotated rx -180 ry 0 rz 180 deg; joints [-27.888, 51.003, -81.346, 31.517, 116.52, 15.313]
  Call Extruder(198.66360)
  MoveL 5776 to (227.77, 35.78, 88.06) mm, rotated rx -180 ry 0 rz 180 deg; joints [-27.834, 51.029, -81.346, 31.452, 116.512, 15.271]
  MoveL 5777 to (227.77, 35.78, 88.06) mm, rotated rx -180 ry 0 rz 180 deg; joints [-27.834, 51.029, -81.346, 31.452, 116.512, 15.271]
  Call Extruder(198.79936)
  MoveL 5778 to (228.02, 35.83, 88.06) mm, rotated rx -180 ry 0 rz 180 deg; joints [-27.78, 51.055, -81.346, 31.387, 116.504, 15.23]
  MoveL 5779 to (228.02, 35.83, 88.06) mm, rotated rx -180 ry 0 rz 180 deg; joints [-27.78, 51.055, -81.346, 31.387, 116.504, 15.23]
  Call Extruder(198.93573)
  MoveL 5780 to (228.27, 35.88, 88.06) mm, rotated rx -180 ry 0 rz 180 deg; joints [-27.726, 51.081, -81.346, 31.322, 116.496, 15.189]
  MoveL 5781 to (228.27, 35.88, 88.06) mm, rotated rx -180 ry 0 rz 180 deg; joints [-27.726, 51.081, -81.346, 31.322, 116.496, 15.189]
  Call Extruder(199.07271)
  MoveL 5782 to (228.52, 35.93, 88.06) mm, rotated rx 180 ry 0 rz 180 deg; joints [-27.673, 51.107, -81.346, 31.258, 116.488, 15.148]
  MoveL 5783 to (228.52, 35.93, 88.06) mm, rotated rx 180 ry 0 rz 180 deg; joints [-27.673, 51.107, -81.346, 31.258, 116.488, 15.148]
  Call Extruder(199.21030)
  MoveL 5784 to (228.77, 35.98, 88.06) mm, rotated rx 180 ry 0 rz 180 deg; joints [-27.62, 51.133, -81.345, 31.194, 116.479, 15.108]
  MoveL 5785 to (228.77, 35.98, 88.06) mm, rotated rx 180 ry 0 rz 180 deg; joints [-27.62, 51.133, -81.345, 31.194, 116.479, 15.108]
  Call Extruder(199.32402)
  MoveL 5786 to (228.97, 36.03, 88.06) mm, rotated rx 180 ry 0 rz -180 deg; joints [-27.579, 51.154, -81.345, 31.144, 116.471, 15.075]
  MoveL 5787 to (228.97, 36.03, 88.06) mm, rotated rx 180 ry 0 rz -180 deg; joints [-27.579, 51.154, -81.345, 31.144, 116.471, 15.075]
  Call Extruder(199.43819)
  MoveL 5788 to (229.18, 36.07, 88.06) mm, rotated rx 180 ry 0 rz 180 deg; joints [-27.539, 51.176, -81.345, 31.095, 116.463, 15.043]
  MoveL 5789 to (229.18, 36.07, 88.06) mm, rotated rx 180 ry 0 rz 180 deg; joints [-27.539, 51.176, -81.345, 31.095, 116.463, 15.043]
  Call Extruder(199.55281)
  MoveL 5790 to (229.38, 36.12, 88.06) mm, rotated rx -180 ry 0 rz 180 deg; joints [-27.499, 51.197, -81.345, 31.046, 116.454, 15.012]
  MoveL 5791 to (229.38, 36.12, 88.06) mm, rotated rx -180 ry 0 rz 180 deg; joints [-27.499, 51.197, -81.345, 31.046, 116.454, 15.012]
  Call Extruder(199.66788)
  MoveL 5792 to (229.59, 36.16, 88.06) mm, rotated rx -180 ry 0 rz 180 deg; joints [-27.458, 51.219, -81.345, 30.997, 116.446, 14.98]
  MoveL 5793 to (229.59, 36.16, 88.06) mm, rotated rx -180 ry 0 rz 180 deg; joints [-27.458, 51.219, -81.345, 30.997, 116.446, 14.98]
  Call Extruder(199.79012)
  MoveL 5794 to (229.8, 36.22, 88.06) mm, rotated rx 180 ry 0 rz 180 deg; joints [-27.423, 51.242, -81.344, 30.953, 116.436, 14.949]
  MoveL 5795 to (229.8, 36.22, 88.06) mm, rotated rx 180 ry 0 rz 180 deg; joints [-27.423, 51.242, -81.344, 30.953, 116.436, 14.949]
  Call Extruder(199.91978)
  MoveL 5796 to (230.02, 36.28, 88.06) mm, rotated rx 180 ry 0 rz 180 deg; joints [-27.392, 51.266, -81.344, 30.913, 116.422, 14.92]
  MoveL 5797 to (230.02, 36.28, 88.06) mm, rotated rx 180 ry 0 rz 180 deg; joints [-27.392, 51.266, -81.344, 30.913, 116.422, 14.92]
  Call Extruder(200.05001)
  MoveL 5798 to (230.25, 36.35, 88.06) mm, rotated rx 180 ry 0 rz 180 deg; joints [-27.361, 51.291, -81.344, 30.874, 116.409, 14.891]
  MoveL 5799 to (230.25, 36.35, 88.06) mm, rotated rx 180 ry 0 rz 180 deg; joints [-27.361, 51.291, -81.344, 30.874, 116.409, 14.891]
  Call Extruder(200.18081)
  MoveL 5800 to (230.47, 36.42, 88.06) mm, rotated rx -180 ry 0 rz 180 deg; joints [-27.33, 51.315, -81.343, 30.833, 116.396, 14.862]
  MoveL 5801 to (230.47, 36.42, 88.06) mm, rotated rx -180 ry 0 rz 180 deg; joints [-27.33, 51.315, -81.343, 30.833, 116.396, 14.862]
  Call Extruder(200.31217)
  MoveL 5802 to (230.69, 36.49, 88.06) mm, rotated rx -180 ry 0 rz 180 deg; joints [-27.299, 51.34, -81.343, 30.794, 116.382, 14.833]
  MoveL 5803 to (230.69, 36.49, 88.06) mm, rotated rx -180 ry 0 rz 180 deg; joints [-27.299, 51.34, -81.343, 30.794, 116.382, 14.833]
  Call Extruder(200.40859)
  MoveL 5804 to (230.86, 36.54, 88.06) mm, rotated rx 180 ry 0 rz 180 deg; joints [-27.28, 51.358, -81.343, 30.768, 116.371, 14.813]
  MoveL 5805 to (230.86, 36.54, 88.06) mm, rotated rx 180 ry 0 rz 180 deg; joints [-27.28, 51.358, -81.343, 30.768, 116.371, 14.813]
  Call Extruder(200.52476)
  MoveL 5806 to (231.05, 36.6, 88.06) mm, rotated rx -180 ry 0 rz 180 deg; joints [-27.256, 51.379, -81.342, 30.737, 116.359, 14.789]
  MoveL 5807 to (231.05, 36.6, 88.06) mm, rotated rx -180 ry 0 rz 180 deg; joints [-27.256, 51.379, -81.342, 30.737, 116.359, 14.789]
  Call Extruder(200.64140)
  MoveL 5808 to (231.25, 36.67, 88.06) mm, rotated rx -180 ry 0 rz 180 deg; joints [-27.232, 51.401, -81.342, 30.706, 116.346, 14.765]
  MoveL 5809 to (231.25, 36.67, 88.06) mm, rotated rx -180 ry 0 rz 180 deg; joints [-27.232, 51.401, -81.342, 30.706, 116.346, 14.765]
  Call Extruder(200.75852)
  MoveL 5810 to (231.44, 36.73, 88.06) mm, rotated rx 180 ry 0 rz 180 deg; joints [-27.209, 51.422, -81.341, 30.675, 116.333, 14.742]
  MoveL 5811 to (231.44, 36.73, 88.06) mm, rotated rx 180 ry 0 rz 180 deg; joints [-27.209, 51.422, -81.341, 30.675, 116.333, 14.742]
  Call Extruder(200.87612)
  MoveL 5812 to (231.64, 36.79, 88.06) mm, rotated rx 180 ry 0 rz -180 deg; joints [-27.185, 51.444, -81.341, 30.644, 116.32, 14.718]
  MoveL 5813 to (231.64, 36.79, 88.06) mm, rotated rx 180 ry 0 rz -180 deg; joints [-27.185, 51.444, -81.341, 30.644, 116.32, 14.718]
  Call Extruder(201.05807)
  MoveL 5814 to (231.93, 36.91, 88.06) mm, rotated rx 180 ry 0 rz -180 deg; joints [-27.167, 51.477, -81.34, 30.616, 116.296, 14.69]
  MoveL 5815 to (231.93, 36.91, 88.06) mm, rotated rx 180 ry 0 rz -180 deg; joints [-27.167, 51.477, -81.34, 30.616, 116.296, 14.69]
  Call Extruder(201.24079)
  MoveL 5816 to (232.22, 37.04, 88.06) mm, rotated rx 180 ry 0 rz 180 deg; joints [-27.149, 51.51, -81.34, 30.588, 116.271, 14.662]
  MoveL 5817 to (232.22, 37.04, 88.06) mm, rotated rx 180 ry 0 rz 180 deg; joints [-27.149, 51.51, -81.34, 30.588, 116.271, 14.662]
  Call Extruder(201.41121)
  MoveL 5818 to (232.49, 37.15, 88.06) mm, rotated rx 180 ry 0 rz -180 deg; joints [-27.133, 51.541, -81.339, 30.564, 116.247, 14.637]
  MoveL 5819 to (232.49, 37.15, 88.06) mm, rotated rx 180 ry 0 rz -180 deg; joints [-27.133, 51.541, -81.339, 30.564, 116.247, 14.637]
  Call Extruder(201.56921)
  MoveL 5820 to (232.74, 37.26, 88.06) mm, rotated rx -180 ry 0 rz 180 deg; joints [-27.121, 51.57, -81.338, 30.542, 116.225, 14.614]
  MoveL 5821 to (232.74, 37.26, 88.06) mm, rotated rx -180 ry 0 rz 180 deg; joints [-27.121, 51.57, -81.338, 30.542, 116.225, 14.614]
  Call Extruder(201.72781)
  MoveL 5822 to (232.99, 37.36, 88.06) mm, rotated rx -180 ry 0 rz 180 deg; joints [-27.108, 51.599, -81.338, 30.521, 116.203, 14.591]
  MoveL 5823 to (232.99, 37.36, 88.06) mm, rotated rx -180 ry 0 rz 180 deg; joints [-27.108, 51.599, -81.338, 30.521, 116.203, 14.591]
  Call Extruder(201.93398)
  MoveL 5824 to (233.29, 37.54, 88.06) mm, rotated rx -180 ry 0 rz 180 deg; joints [-27.12, 51.636, -81.337, 30.524, 116.168, 14.575]
  MoveL 5825 to (233.29, 37.54, 88.06) mm, rotated rx -180 ry 0 rz 180 deg; joints [-27.12, 51.636, -81.337, 30.524, 116.168, 14.575]
  Call Extruder(202.14092)
  MoveL 5826 to (233.6, 37.71, 88.06) mm, rotated rx 180 ry 0 rz -180 deg; joints [-27.132, 51.673, -81.336, 30.528, 116.132, 14.56]
  MoveL 5827 to (233.6, 37.71, 88.06) mm, rotated rx 180 ry 0 rz -180 deg; joints [-27.132, 51.673, -81.336, 30.528, 116.132, 14.56]
  Call Extruder(202.34865)
  MoveL 5828 to (233.9, 37.89, 88.06) mm, rotated rx -180 ry 0 rz 180 deg; joints [-27.144, 51.71, -81.335, 30.532, 116.096, 14.544]
  MoveL 5829 to (233.9, 37.89, 88.06) mm, rotated rx -180 ry 0 rz 180 deg; joints [-27.144, 51.71, -81.335, 30.532, 116.096, 14.544]
  Call Extruder(202.55715)
  MoveL 5830 to (234.21, 38.06, 88.06) mm, rotated rx -180 ry 0 rz 180 deg; joints [-27.156, 51.747, -81.333, 30.535, 116.06, 14.528]
  MoveL 5831 to (234.21, 38.06, 88.06) mm, rotated rx -180 ry 0 rz 180 deg; joints [-27.156, 51.747, -81.333, 30.535, 116.06, 14.528]
  Call Extruder(202.73669)
  MoveL 5832 to (234.45, 38.24, 88.06) mm, rotated rx 180 ry 0 rz -180 deg; joints [-27.187, 51.778, -81.332, 30.56, 116.024, 14.524]
  MoveL 5833 to (234.45, 38.24, 88.06) mm, rotated rx 180 ry 0 rz -180 deg; joints [-27.187, 51.778, -81.332, 30.56, 116.024, 14.524]
  Call Extruder(203.07011)
  MoveL 5834 to (234.9, 38.57, 88.06) mm, rotated rx 180 ry 0 rz 180 deg; joints [-27.245, 51.836, -81.331, 30.608, 115.958, 14.518]
  MoveL 5835 to (234.9, 38.57, 88.06) mm, rotated rx 180 ry 0 rz 180 deg; joints [-27.245, 51.836, -81.331, 30.608, 115.958, 14.518]
  Call Extruder(203.40471)
  MoveL 5836 to (235.35, 38.9, 88.06) mm, rotated rx -180 ry 0 rz 180 deg; joints [-27.302, 51.895, -81.329, 30.655, 115.892, 14.511]
  Call Extruder(204.23266)
  MoveL 5837 to (236.39, 39.81, 88.06) mm, rotated rx -180 ry 0 rz 180 deg; joints [-27.525, 52.035, -81.323, 30.858, 115.711, 14.532]
  Call Extruder(205.06060)
  MoveL 5838 to (237.3, 40.85, 88.06) mm, rotated rx 180 ry 0 rz 180 deg; joints [-27.851, 52.17, -81.317, 31.174, 115.508, 14.603]
  Call Extruder(205.22791)
  MoveL 5839 to (237.47, 41.07, 88.06) mm, rotated rx -180 ry 0 rz 180 deg; joints [-27.932, 52.197, -81.316, 31.253, 115.464, 14.624]
  MoveL 5840 to (237.47, 41.07, 88.06) mm, rotated rx -180 ry 0 rz 180 deg; joints [-27.932, 52.197, -81.316, 31.253, 115.464, 14.624]
  Call Extruder(205.56133)
  MoveL 5841 to (237.79, 41.52, 88.06) mm, rotated rx -180 ry 0 rz 180 deg; joints [-28.091, 52.249, -81.314, 31.41, 115.377, 14.666]
  MoveL 5842 to (237.79, 41.52, 88.06) mm, rotated rx -180 ry 0 rz 180 deg; joints [-28.091, 52.249, -81.314, 31.41, 115.377, 14.666]
  Call Extruder(205.89358)
  MoveL 5843 to (238.12, 41.98, 88.06) mm, rotated rx 180 ry 0 rz 180 deg; joints [-28.249, 52.302, -81.311, 31.565, 115.29, 14.706]
  MoveL 5844 to (238.12, 41.98, 88.06) mm, rotated rx 180 ry 0 rz 180 deg; joints [-28.249, 52.302, -81.311, 31.565, 115.29, 14.706]
  Call Extruder(206.06099)
  MoveL 5845 to (238.27, 42.22, 88.06) mm, rotated rx -180 ry 0 rz 180 deg; joints [-28.342, 52.327, -81.31, 31.658, 115.244, 14.733]
  MoveL 5846 to (238.27, 42.22, 88.06) mm, rotated rx -180 ry 0 rz 180 deg; joints [-28.342, 52.327, -81.31, 31.658, 115.244, 14.733]
  Call Extruder(206.21452)
  MoveL 5847 to (238.4, 42.44, 88.06) mm, rotated rx 180 ry 0 rz 180 deg; joints [-28.427, 52.35, -81.309, 31.744, 115.201, 14.758]
  MoveL 5848 to (238.4, 42.44, 88.06) mm, rotated rx 180 ry 0 rz 180 deg; joints [-28.427, 52.35, -81.309, 31.744, 115.201, 14.758]
  Call Extruder(206.42306)
  MoveL 5849 to (238.58, 42.75, 88.06) mm, rotated rx 180 ry 0 rz 180 deg; joints [-28.548, 52.381, -81.307, 31.864, 115.143, 14.794]
  MoveL 5850 to (238.58, 42.75, 88.06) mm, rotated rx 180 ry 0 rz 180 deg; joints [-28.548, 52.381, -81.307, 31.864, 115.143, 14.794]
  Call Extruder(206.63087)
  MoveL 5851 to (238.75, 43.06, 88.06) mm, rotated rx -180 ry 0 rz 180 deg; joints [-28.667, 52.413, -81.306, 31.984, 115.084, 14.829]
  MoveL 5852 to (238.75, 43.06, 88.06) mm, rotated rx -180 ry 0 rz 180 deg; joints [-28.667, 52.413, -81.306, 31.984, 115.084, 14.829]
  Call Extruder(206.81346)
  MoveL 5853 to (238.89, 43.33, 88.06) mm, rotated rx 180 ry 0 rz 180 deg; joints [-28.78, 52.439, -81.304, 32.097, 115.031, 14.863]
  MoveL 5854 to (238.89, 43.33, 88.06) mm, rotated rx 180 ry 0 rz 180 deg; joints [-28.78, 52.439, -81.304, 32.097, 115.031, 14.863]
  Call Extruder(206.97148)
  MoveL 5855 to (239, 43.58, 88.06) mm, rotated rx -180 ry 0 rz 180 deg; joints [-28.886, 52.462, -81.303, 32.204, 114.984, 14.897]
  MoveL 5856 to (239, 43.58, 88.06) mm, rotated rx -180 ry 0 rz 180 deg; joints [-28.886, 52.462, -81.303, 32.204, 114.984, 14.897]
  Call Extruder(207.12890)
  MoveL 5857 to (239.11, 43.83, 88.06) mm, rotated rx -180 ry 0 rz 180 deg; joints [-28.991, 52.484, -81.302, 32.311, 114.937, 14.93]
  MoveL 5858 to (239.11, 43.83, 88.06) mm, rotated rx -180 ry 0 rz 180 deg; joints [-28.991, 52.484, -81.302, 32.311, 114.937, 14.93]
  Call Extruder(207.31161)
  MoveL 5859 to (239.22, 44.12, 88.06) mm, rotated rx -180 ry 0 rz 180 deg; joints [-29.116, 52.51, -81.3, 32.437, 114.882, 14.97]
  MoveL 5860 to (239.22, 44.12, 88.06) mm, rotated rx -180 ry 0 rz 180 deg; joints [-29.116, 52.51, -81.3, 32.437, 114.882, 14.97]
  Call Extruder(207.49357)
  MoveL 5861 to (239.35, 44.42, 88.06) mm, rotated rx 180 ry 0 rz 180 deg; joints [-29.24, 52.535, -81.299, 32.562, 114.827, 15.01]
  MoveL 5862 to (239.35, 44.42, 88.06) mm, rotated rx 180 ry 0 rz 180 deg; joints [-29.24, 52.535, -81.299, 32.562, 114.827, 15.01]
  Call Extruder(207.64090)
  MoveL 5863 to (239.44, 44.66, 88.06) mm, rotated rx 180 ry 0 rz 180 deg; joints [-29.343, 52.556, -81.297, 32.666, 114.782, 15.043]
  MoveL 5864 to (239.44, 44.66, 88.06) mm, rotated rx 180 ry 0 rz 180 deg; joints [-29.343, 52.556, -81.297, 32.666, 114.782, 15.043]
  Call Extruder(207.75414)
  MoveL 5865 to (239.5, 44.85, 88.06) mm, rotated rx 180 ry 0 rz 180 deg; joints [-29.428, 52.571, -81.297, 32.752, 114.747, 15.071]
  MoveL 5866 to (239.5, 44.85, 88.06) mm, rotated rx 180 ry 0 rz 180 deg; joints [-29.428, 52.571, -81.297, 32.752, 114.747, 15.071]
  Call Extruder(207.86693)
  MoveL 5867 to (239.56, 45.03, 88.06) mm, rotated rx -180 ry 0 rz 180 deg; joints [-29.512, 52.586, -81.296, 32.837, 114.711, 15.099]
  MoveL 5868 to (239.56, 45.03, 88.06) mm, rotated rx -180 ry 0 rz 180 deg; joints [-29.512, 52.586, -81.296, 32.837, 114.711, 15.099]
  Call Extruder(207.97927)
  MoveL 5869 to (239.62, 45.22, 88.06) mm, rotated rx 180 ry 0 rz 180 deg; joints [-29.596, 52.601, -81.295, 32.923, 114.676, 15.126]
  MoveL 5870 to (239.62, 45.22, 88.06) mm, rotated rx 180 ry 0 rz 180 deg; joints [-29.596, 52.601, -81.295, 32.923, 114.676, 15.126]
  Call Extruder(208.09117)
  MoveL 5871 to (239.68, 45.41, 88.06) mm, rotated rx 180 ry 0 rz 180 deg; joints [-29.679, 52.616, -81.294, 33.007, 114.641, 15.154]
  MoveL 5872 to (239.68, 45.41, 88.06) mm, rotated rx 180 ry 0 rz 180 deg; joints [-29.679, 52.616, -81.294, 33.007, 114.641, 15.154]
  Call Extruder(208.21257)
  MoveL 5873 to (239.75, 45.62, 88.06) mm, rotated rx -180 ry 0 rz 180 deg; joints [-29.77, 52.633, -81.293, 33.1, 114.602, 15.184]
  MoveL 5874 to (239.75, 45.62, 88.06) mm, rotated rx -180 ry 0 rz 180 deg; joints [-29.77, 52.633, -81.293, 33.1, 114.602, 15.184]
  Call Extruder(208.34336)
  MoveL 5875 to (239.82, 45.84, 88.06) mm, rotated rx 180 ry 0 rz 180 deg; joints [-29.871, 52.65, -81.292, 33.201, 114.56, 15.217]
  MoveL 5876 to (239.82, 45.84, 88.06) mm, rotated rx 180 ry 0 rz 180 deg; joints [-29.871, 52.65, -81.292, 33.201, 114.56, 15.217]
  Call Extruder(208.47359)
  MoveL 5877 to (239.88, 46.06, 88.06) mm, rotated rx 180 ry 0 rz 180 deg; joints [-29.97, 52.668, -81.291, 33.302, 114.518, 15.249]
  MoveL 5878 to (239.88, 46.06, 88.06) mm, rotated rx 180 ry 0 rz 180 deg; joints [-29.97, 52.668, -81.291, 33.302, 114.518, 15.249]
  Call Extruder(208.60325)
  MoveL 5879 to (239.95, 46.29, 88.06) mm, rotated rx -180 ry 0 rz 180 deg; joints [-30.069, 52.686, -81.289, 33.403, 114.477, 15.282]
  MoveL 5880 to (239.95, 46.29, 88.06) mm, rotated rx -180 ry 0 rz 180 deg; joints [-30.069, 52.686, -81.289, 33.403, 114.477, 15.282]
  Call Extruder(208.73235)
  MoveL 5881 to (240.02, 46.51, 88.06) mm, rotated rx 180 ry 0 rz 180 deg; joints [-30.168, 52.703, -81.288, 33.503, 114.435, 15.314]
  MoveL 5882 to (240.02, 46.51, 88.06) mm, rotated rx 180 ry 0 rz 180 deg; joints [-30.168, 52.703, -81.288, 33.503, 114.435, 15.314]
  Call Extruder(208.84740)
  MoveL 5883 to (240.06, 46.72, 88.06) mm, rotated rx -180 ry 0 rz 180 deg; joints [-30.263, 52.718, -81.287, 33.6, 114.397, 15.346]
  MoveL 5884 to (240.06, 46.72, 88.06) mm, rotated rx -180 ry 0 rz 180 deg; joints [-30.263, 52.718, -81.287, 33.6, 114.397, 15.346]
  Call Extruder(208.96201)
  MoveL 5885 to (240.11, 46.92, 88.06) mm, rotated rx -180 ry 0 rz 180 deg; joints [-30.358, 52.733, -81.286, 33.696, 114.359, 15.378]
  MoveL 5886 to (240.11, 46.92, 88.06) mm, rotated rx -180 ry 0 rz 180 deg; joints [-30.358, 52.733, -81.286, 33.696, 114.359, 15.378]
  Call Extruder(209.07616)
  MoveL 5887 to (240.15, 47.12, 88.06) mm, rotated rx -180 ry 0 rz 180 deg; joints [-30.453, 52.747, -81.286, 33.793, 114.32, 15.41]
  MoveL 5888 to (240.15, 47.12, 88.06) mm, rotated rx -180 ry 0 rz 180 deg; joints [-30.453, 52.747, -81.286, 33.793, 114.32, 15.41]
  Call Extruder(209.18985)
  MoveL 5889 to (240.2, 47.33, 88.06) mm, rotated rx -180 ry 0 rz 180 deg; joints [-30.548, 52.762, -81.285, 33.889, 114.282, 15.441]
  MoveL 5890 to (240.2, 47.33, 88.06) mm, rotated rx -180 ry 0 rz 180 deg; joints [-30.548, 52.762, -81.285, 33.889, 114.282, 15.441]
  Call Extruder(209.31526)
  MoveL 5891 to (240.24, 47.55, 88.06) mm, rotated rx -180 ry 0 rz 180 deg; joints [-30.653, 52.778, -81.283, 33.995, 114.24, 15.476]
  MoveL 5892 to (240.24, 47.55, 88.06) mm, rotated rx -180 ry 0 rz 180 deg; joints [-30.653, 52.778, -81.283, 33.995, 114.24, 15.476]
  Call Extruder(209.45224)
  MoveL 5893 to (240.29, 47.8, 88.06) mm, rotated rx -180 ry 0 rz 180 deg; joints [-30.768, 52.796, -81.282, 34.113, 114.194, 15.515]
  MoveL 5894 to (240.29, 47.8, 88.06) mm, rotated rx -180 ry 0 rz 180 deg; joints [-30.768, 52.796, -81.282, 34.113, 114.194, 15.515]
  Call Extruder(209.58861)
  MoveL 5895 to (240.34, 48.05, 88.06) mm, rotated rx -180 ry 0 rz 180 deg; joints [-30.884, 52.813, -81.281, 34.23, 114.147, 15.553]
  MoveL 5896 to (240.34, 48.05, 88.06) mm, rotated rx -180 ry 0 rz 180 deg; joints [-30.884, 52.813, -81.281, 34.23, 114.147, 15.553]
  Call Extruder(209.72437)
  MoveL 5897 to (240.39, 48.3, 88.06) mm, rotated rx 180 ry 0 rz 180 deg; joints [-30.999, 52.831, -81.28, 34.347, 114.101, 15.591]
  MoveL 5898 to (240.39, 48.3, 88.06) mm, rotated rx 180 ry 0 rz 180 deg; joints [-30.999, 52.831, -81.28, 34.347, 114.101, 15.591]
  Call Extruder(209.85951)
  MoveL 5899 to (240.44, 48.55, 88.06) mm, rotated rx -180 ry 0 rz 180 deg; joints [-31.114, 52.848, -81.279, 34.464, 114.054, 15.629]
  MoveL 5900 to (240.44, 48.55, 88.06) mm, rotated rx -180 ry 0 rz 180 deg; joints [-31.114, 52.848, -81.279, 34.464, 114.054, 15.629]
  Call Extruder(209.99405)
  MoveL 5901 to (240.49, 48.8, 88.06) mm, rotated rx -180 ry 0 rz 180 deg; joints [-31.228, 52.866, -81.277, 34.579, 114.008, 15.666]
  MoveL 5902 to (240.49, 48.8, 88.06) mm, rotated rx -180 ry 0 rz 180 deg; joints [-31.228, 52.866, -81.277, 34.579, 114.008, 15.666]
  Call Extruder(210.12798)
  MoveL 5903 to (240.54, 49.05, 88.06) mm, rotated rx 180 ry 0 rz 180 deg; joints [-31.342, 52.884, -81.276, 34.694, 113.961, 15.703]
  MoveL 5904 to (240.54, 49.05, 88.06) mm, rotated rx 180 ry 0 rz 180 deg; joints [-31.342, 52.884, -81.276, 34.694, 113.961, 15.703]
  Call Extruder(210.27584)
  MoveL 5905 to (240.59, 49.33, 88.06) mm, rotated rx 180 ry 0 rz 180 deg; joints [-31.47, 52.903, -81.275, 34.824, 113.91, 15.745]
  MoveL 5906 to (240.59, 49.33, 88.06) mm, rotated rx 180 ry 0 rz 180 deg; joints [-31.47, 52.903, -81.275, 34.824, 113.91, 15.745]
  Call Extruder(210.43759)
  MoveL 5907 to (240.64, 49.63, 88.06) mm, rotated rx -180 ry 0 rz 180 deg; joints [-31.612, 52.924, -81.273, 34.968, 113.853, 15.792]
  MoveL 5908 to (240.64, 49.63, 88.06) mm, rotated rx -180 ry 0 rz 180 deg; joints [-31.612, 52.924, -81.273, 34.968, 113.853, 15.792]
  Call Extruder(210.59860)
  MoveL 5909 to (240.69, 49.94, 88.06) mm, rotated rx -180 ry 0 rz 180 deg; joints [-31.755, 52.944, -81.272, 35.112, 113.796, 15.839]
  MoveL 5910 to (240.69, 49.94, 88.06) mm, rotated rx -180 ry 0 rz 180 deg; joints [-31.755, 52.944, -81.272, 35.112, 113.796, 15.839]
  Call Extruder(210.75889)
  MoveL 5911 to (240.73, 50.24, 88.06) mm, rotated rx 180 ry 0 rz 180 deg; joints [-31.895, 52.965, -81.27, 35.254, 113.739, 15.884]
  MoveL 5912 to (240.73, 50.24, 88.06) mm, rotated rx 180 ry 0 rz 180 deg; joints [-31.895, 52.965, -81.27, 35.254, 113.739, 15.884]
  Call Extruder(210.91845)
  MoveL 5913 to (240.78, 50.55, 88.06) mm, rotated rx -180 ry 0 rz 180 deg; joints [-32.036, 52.986, -81.269, 35.397, 113.682, 15.929]
  MoveL 5914 to (240.78, 50.55, 88.06) mm, rotated rx -180 ry 0 rz 180 deg; joints [-32.036, 52.986, -81.269, 35.397, 113.682, 15.929]
  Call Extruder(211.07728)
  MoveL 5915 to (240.83, 50.86, 88.06) mm, rotated rx 180 ry 0 rz 180 deg; joints [-32.176, 53.007, -81.267, 35.538, 113.625, 15.974]
  MoveL 5916 to (240.83, 50.86, 88.06) mm, rotated rx 180 ry 0 rz 180 deg; joints [-32.176, 53.007, -81.267, 35.538, 113.625, 15.974]
  Call Extruder(211.25596)
  MoveL 5917 to (240.88, 51.2, 88.06) mm, rotated rx -180 ry 0 rz 180 deg; joints [-32.337, 53.03, -81.265, 35.7, 113.561, 16.026]
  MoveL 5918 to (240.88, 51.2, 88.06) mm, rotated rx -180 ry 0 rz 180 deg; joints [-32.337, 53.03, -81.265, 35.7, 113.561, 16.026]
  Call Extruder(211.45440)
  MoveL 5919 to (240.93, 51.59, 88.06) mm, rotated rx 180 ry 0 rz 180 deg; joints [-32.518, 53.055, -81.263, 35.883, 113.489, 16.084]
  MoveL 5920 to (240.93, 51.59, 88.06) mm, rotated rx 180 ry 0 rz 180 deg; joints [-32.518, 53.055, -81.263, 35.883, 113.489, 16.084]
  Call Extruder(211.65197)
  MoveL 5921 to (240.97, 51.98, 88.06) mm, rotated rx 180 ry 0 rz 180 deg; joints [-32.697, 53.081, -81.261, 36.064, 113.417, 16.141]
  MoveL 5922 to (240.97, 51.98, 88.06) mm, rotated rx 180 ry 0 rz 180 deg; joints [-32.697, 53.081, -81.261, 36.064, 113.417, 16.141]
  Call Extruder(211.84868)
  MoveL 5923 to (241.02, 52.37, 88.06) mm, rotated rx -180 ry 0 rz 180 deg; joints [-32.876, 53.106, -81.259, 36.244, 113.345, 16.198]
  MoveL 5924 to (241.02, 52.37, 88.06) mm, rotated rx -180 ry 0 rz 180 deg; joints [-32.876, 53.106, -81.259, 36.244, 113.345, 16.198]
  Call Extruder(212.04452)
  MoveL 5925 to (241.06, 52.75, 88.06) mm, rotated rx -180 ry 0 rz -180 deg; joints [-33.055, 53.132, -81.257, 36.423, 113.273, 16.254]
  MoveL 5926 to (241.06, 52.75, 88.06) mm, rotated rx -180 ry 0 rz -180 deg; joints [-33.055, 53.132, -81.257, 36.423, 113.273, 16.254]
  Call Extruder(212.33996)
  MoveL 5927 to (241.11, 53.34, 88.06) mm, rotated rx -180 ry 0 rz 180 deg; joints [-33.331, 53.169, -81.254, 36.702, 113.163, 16.342]
  MoveL 5928 to (241.11, 53.34, 88.06) mm, rotated rx -180 ry 0 rz 180 deg; joints [-33.331, 53.169, -81.254, 36.702, 113.163, 16.342]
  Call Extruder(212.63406)
  MoveL 5929 to (241.16, 53.93, 88.06) mm, rotated rx 180 ry 0 rz 180 deg; joints [-33.606, 53.206, -81.251, 36.978, 113.053, 16.428]
  MoveL 5930 to (241.16, 53.93, 88.06) mm, rotated rx 180 ry 0 rz 180 deg; joints [-33.606, 53.206, -81.251, 36.978, 113.053, 16.428]
  Call Extruder(212.92684)
  MoveL 5931 to (241.2, 54.52, 88.06) mm, rotated rx -180 ry 0 rz 180 deg; joints [-33.878, 53.244, -81.248, 37.252, 112.944, 16.512]
  MoveL 5932 to (241.2, 54.52, 88.06) mm, rotated rx -180 ry 0 rz 180 deg; joints [-33.878, 53.244, -81.248, 37.252, 112.944, 16.512]
  Call Extruder(213.50029)
  MoveL 5933 to (241.25, 55.68, 88.06) mm, rotated rx -180 ry 0 rz 180 deg; joints [-34.425, 53.314, -81.242, 37.8, 112.727, 16.682]
  MoveL 5934 to (241.25, 55.68, 88.06) mm, rotated rx -180 ry 0 rz 180 deg; joints [-34.425, 53.314, -81.242, 37.8, 112.727, 16.682]
  Call Extruder(214.21412)
  MoveL 5935 to (241.29, 57.14, 88.06) mm, rotated rx -180 ry 0 rz -180 deg; joints [-35.104, 53.402, -81.234, 38.48, 112.455, 16.889]
  Call Extruder(256.27901)
  MoveL 5936 to (241.29, 142.86, 88.06) mm, rotated rx -180 ry 0 rz -180 deg; joints [-60.361, 59.5, -79.834, 61.919, 99.895, 17.853]
  Call Extruder(256.70743)
  MoveL 5937 to (241.27, 143.74, 88.06) mm, rotated rx 180 ry 0 rz -180 deg; joints [-60.516, 59.564, -79.808, 62.055, 99.806, 17.799]
  MoveL 5938 to (241.27, 143.74, 88.06) mm, rotated rx 180 ry 0 rz -180 deg; joints [-60.516, 59.564, -79.808, 62.055, 99.806, 17.799]
  Call Extruder(257.28088)
  MoveL 5939 to (241.22, 144.9, 88.06) mm, rotated rx -180 ry 0 rz -180 deg; joints [-60.726, 59.648, -79.774, 62.241, 99.686, 17.727]
  MoveL 5940 to (241.22, 144.9, 88.06) mm, rotated rx -180 ry 0 rz -180 deg; joints [-60.726, 59.648, -79.774, 62.241, 99.686, 17.727]
  Call Extruder(257.71522)
  MoveL 5941 to (241.18, 145.77, 88.06) mm, rotated rx 180 ry 0 rz 180 deg; joints [-60.887, 59.711, -79.748, 62.383, 99.596, 17.674]
  MoveL 5942 to (241.18, 145.77, 88.06) mm, rotated rx 180 ry 0 rz 180 deg; joints [-60.887, 59.711, -79.748, 62.383, 99.596, 17.674]
  Call Extruder(258.00933)
  MoveL 5943 to (241.13, 146.36, 88.06) mm, rotated rx -180 ry 0 rz 180 deg; joints [-61, 59.752, -79.731, 62.482, 99.535, 17.639]
  MoveL 5944 to (241.13, 146.36, 88.06) mm, rotated rx -180 ry 0 rz 180 deg; joints [-61, 59.752, -79.731, 62.482, 99.535, 17.639]
  Call Extruder(258.30477)
  MoveL 5945 to (241.09, 146.95, 88.06) mm, rotated rx -180 ry 0 rz -180 deg; joints [-61.111, 59.794, -79.714, 62.581, 99.474, 17.604]
  MoveL 5946 to (241.09, 146.95, 88.06) mm, rotated rx -180 ry 0 rz -180 deg; joints [-61.111, 59.794, -79.714, 62.581, 99.474, 17.604]
  Call Extruder(258.55103)
  MoveL 5947 to (241.04, 147.44, 88.06) mm, rotated rx 180 ry 0 rz 180 deg; joints [-61.205, 59.828, -79.7, 62.665, 99.423, 17.575]
  MoveL 5948 to (241.04, 147.44, 88.06) mm, rotated rx 180 ry 0 rz 180 deg; joints [-61.205, 59.828, -79.7, 62.665, 99.423, 17.575]
  Call Extruder(258.74773)
  MoveL 5949 to (240.99, 147.83, 88.06) mm, rotated rx 180 ry 0 rz 180 deg; joints [-61.282, 59.855, -79.688, 62.734, 99.383, 17.553]
  MoveL 5950 to (240.99, 147.83, 88.06) mm, rotated rx 180 ry 0 rz 180 deg; joints [-61.282, 59.855, -79.688, 62.734, 99.383, 17.553]
  Call Extruder(258.94530)
  MoveL 5951 to (240.95, 148.22, 88.06) mm, rotated rx 180 ry 0 rz 180 deg; joints [-61.359, 59.881, -79.677, 62.802, 99.342, 17.531]
  MoveL 5952 to (240.95, 148.22, 88.06) mm, rotated rx 180 ry 0 rz 180 deg; joints [-61.359, 59.881, -79.677, 62.802, 99.342, 17.531]
  Call Extruder(259.14375)
  MoveL 5953 to (240.9, 148.6, 88.06) mm, rotated rx 180 ry 0 rz -180 deg; joints [-61.436, 59.908, -79.666, 62.871, 99.302, 17.509]
  MoveL 5954 to (240.9, 148.6, 88.06) mm, rotated rx 180 ry 0 rz -180 deg; joints [-61.436, 59.908, -79.666, 62.871, 99.302, 17.509]
  Call Extruder(259.34306)
  MoveL 5955 to (240.86, 148.99, 88.06) mm, rotated rx -180 ry 0 rz -180 deg; joints [-61.512, 59.935, -79.654, 62.939, 99.261, 17.486]
  MoveL 5956 to (240.86, 148.99, 88.06) mm, rotated rx -180 ry 0 rz -180 deg; joints [-61.512, 59.935, -79.654, 62.939, 99.261, 17.486]
  Call Extruder(259.50189)
  MoveL 5957 to (240.81, 149.3, 88.06) mm, rotated rx 180 ry 0 rz 180 deg; joints [-61.575, 59.956, -79.645, 62.996, 99.229, 17.469]
  MoveL 5958 to (240.81, 149.3, 88.06) mm, rotated rx 180 ry 0 rz 180 deg; joints [-61.575, 59.956, -79.645, 62.996, 99.229, 17.469]
  Call Extruder(259.66145)
  MoveL 5959 to (240.76, 149.6, 88.06) mm, rotated rx -180 ry 0 rz 180 deg; joints [-61.639, 59.976, -79.637, 63.053, 99.197, 17.453]
  MoveL 5960 to (240.76, 149.6, 88.06) mm, rotated rx -180 ry 0 rz 180 deg; joints [-61.639, 59.976, -79.637, 63.053, 99.197, 17.453]
  Call Extruder(259.82174)
  MoveL 5961 to (240.71, 149.91, 88.06) mm, rotated rx -180 ry 0 rz 180 deg; joints [-61.702, 59.997, -79.628, 63.11, 99.164, 17.436]
  MoveL 5962 to (240.71, 149.91, 88.06) mm, rotated rx -180 ry 0 rz 180 deg; joints [-61.702, 59.997, -79.628, 63.11, 99.164, 17.436]
  Call Extruder(259.98276)
  MoveL 5963 to (240.66, 150.21, 88.06) mm, rotated rx -180 ry 0 rz 180 deg; joints [-61.765, 60.017, -79.619, 63.167, 99.132, 17.419]
  MoveL 5964 to (240.66, 150.21, 88.06) mm, rotated rx -180 ry 0 rz 180 deg; joints [-61.765, 60.017, -79.619, 63.167, 99.132, 17.419]
  Call Extruder(260.14450)
  MoveL 5965 to (240.61, 150.52, 88.06) mm, rotated rx 180 ry 0 rz 180 deg; joints [-61.828, 60.038, -79.61, 63.223, 99.1, 17.402]
  MoveL 5966 to (240.61, 150.52, 88.06) mm, rotated rx 180 ry 0 rz 180 deg; joints [-61.828, 60.038, -79.61, 63.223, 99.1, 17.402]
  Call Extruder(260.30697)
  MoveL 5967 to (240.56, 150.83, 88.06) mm, rotated rx -180 ry 0 rz 180 deg; joints [-61.891, 60.058, -79.601, 63.28, 99.068, 17.385]
  MoveL 5968 to (240.56, 150.83, 88.06) mm, rotated rx -180 ry 0 rz 180 deg; joints [-61.891, 60.058, -79.601, 63.28, 99.068, 17.385]
  Call Extruder(260.44090)
  MoveL 5969 to (240.52, 151.07, 88.06) mm, rotated rx -180 ry 0 rz 180 deg; joints [-61.944, 60.075, -79.594, 63.328, 99.041, 17.372]
  MoveL 5970 to (240.52, 151.07, 88.06) mm, rotated rx -180 ry 0 rz 180 deg; joints [-61.944, 60.075, -79.594, 63.328, 99.041, 17.372]
  Call Extruder(260.57544)
  MoveL 5971 to (240.47, 151.32, 88.06) mm, rotated rx -180 ry 0 rz 180 deg; joints [-61.998, 60.091, -79.587, 63.377, 99.015, 17.358]
  MoveL 5972 to (240.47, 151.32, 88.06) mm, rotated rx -180 ry 0 rz 180 deg; joints [-61.998, 60.091, -79.587, 63.377, 99.015, 17.358]
  Call Extruder(260.71058)
  MoveL 5973 to (240.42, 151.57, 88.06) mm, rotated rx -180 ry 0 rz 180 deg; joints [-62.052, 60.108, -79.58, 63.426, 98.988, 17.345]
  MoveL 5974 to (240.42, 151.57, 88.06) mm, rotated rx -180 ry 0 rz 180 deg; joints [-62.052, 60.108, -79.58, 63.426, 98.988, 17.345]
  Call Extruder(260.84634)
  MoveL 5975 to (240.37, 151.82, 88.06) mm, rotated rx 180 ry 0 rz 180 deg; joints [-62.105, 60.124, -79.572, 63.474, 98.962, 17.332]
  MoveL 5976 to (240.37, 151.82, 88.06) mm, rotated rx 180 ry 0 rz 180 deg; joints [-62.105, 60.124, -79.572, 63.474, 98.962, 17.332]
  Call Extruder(260.98271)
  MoveL 5977 to (240.32, 152.07, 88.06) mm, rotated rx 180 ry 0 rz 180 deg; joints [-62.159, 60.14, -79.565, 63.522, 98.935, 17.319]
  MoveL 5978 to (240.32, 152.07, 88.06) mm, rotated rx 180 ry 0 rz 180 deg; joints [-62.159, 60.14, -79.565, 63.522, 98.935, 17.319]
  Call Extruder(261.11969)
  MoveL 5979 to (240.27, 152.32, 88.06) mm, rotated rx 180 ry 0 rz 180 deg; joints [-62.212, 60.157, -79.558, 63.57, 98.909, 17.305]
  MoveL 5980 to (240.27, 152.32, 88.06) mm, rotated rx 180 ry 0 rz 180 deg; joints [-62.212, 60.157, -79.558, 63.57, 98.909, 17.305]
  Call Extruder(261.25727)
  MoveL 5981 to (240.22, 152.57, 88.06) mm, rotated rx -180 ry 0 rz 180 deg; joints [-62.265, 60.173, -79.551, 63.619, 98.882, 17.292]
  MoveL 5982 to (240.22, 152.57, 88.06) mm, rotated rx -180 ry 0 rz 180 deg; joints [-62.265, 60.173, -79.551, 63.619, 98.882, 17.292]
  Call Extruder(261.37097)
  MoveL 5983 to (240.17, 152.77, 88.06) mm, rotated rx -180 ry 0 rz 180 deg; joints [-62.31, 60.186, -79.545, 63.659, 98.861, 17.281]
  MoveL 5984 to (240.17, 152.77, 88.06) mm, rotated rx -180 ry 0 rz 180 deg; joints [-62.31, 60.186, -79.545, 63.659, 98.861, 17.281]
  Call Extruder(261.48512)
  MoveL 5985 to (240.13, 152.98, 88.06) mm, rotated rx 180 ry 0 rz 180 deg; joints [-62.355, 60.2, -79.539, 63.7, 98.839, 17.27]
  MoveL 5986 to (240.13, 152.98, 88.06) mm, rotated rx 180 ry 0 rz 180 deg; joints [-62.355, 60.2, -79.539, 63.7, 98.839, 17.27]
  Call Extruder(261.59972)
  MoveL 5987 to (240.08, 153.18, 88.06) mm, rotated rx -180 ry 0 rz 180 deg; joints [-62.399, 60.213, -79.533, 63.74, 98.817, 17.259]
  MoveL 5988 to (240.08, 153.18, 88.06) mm, rotated rx -180 ry 0 rz 180 deg; joints [-62.399, 60.213, -79.533, 63.74, 98.817, 17.259]
  Call Extruder(261.71478)
  MoveL 5989 to (240.04, 153.39, 88.06) mm, rotated rx 180 ry 0 rz 180 deg; joints [-62.444, 60.226, -79.527, 63.78, 98.795, 17.248]
  MoveL 5990 to (240.04, 153.39, 88.06) mm, rotated rx 180 ry 0 rz 180 deg; joints [-62.444, 60.226, -79.527, 63.78, 98.795, 17.248]
  Call Extruder(261.83700)
  MoveL 5991 to (239.98, 153.6, 88.06) mm, rotated rx -180 ry 0 rz -180 deg; joints [-62.493, 60.24, -79.521, 63.825, 98.772, 17.238]
  MoveL 5992 to (239.98, 153.6, 88.06) mm, rotated rx -180 ry 0 rz -180 deg; joints [-62.493, 60.24, -79.521, 63.825, 98.772, 17.238]
  Call Extruder(261.96666)
  MoveL 5993 to (239.92, 153.82, 88.06) mm, rotated rx 180 ry 0 rz 180 deg; joints [-62.547, 60.254, -79.515, 63.874, 98.747, 17.228]
  MoveL 5994 to (239.92, 153.82, 88.06) mm, rotated rx 180 ry 0 rz 180 deg; joints [-62.547, 60.254, -79.515, 63.874, 98.747, 17.228]
  Call Extruder(262.09688)
  MoveL 5995 to (239.85, 154.05, 88.06) mm, rotated rx -180 ry 0 rz -180 deg; joints [-62.601, 60.267, -79.508, 63.924, 98.723, 17.217]
  MoveL 5996 to (239.85, 154.05, 88.06) mm, rotated rx -180 ry 0 rz -180 deg; joints [-62.601, 60.267, -79.508, 63.924, 98.723, 17.217]
  Call Extruder(262.22767)
  MoveL 5997 to (239.78, 154.27, 88.06) mm, rotated rx 180 ry 0 rz -180 deg; joints [-62.654, 60.281, -79.502, 63.973, 98.698, 17.207]
  MoveL 5998 to (239.78, 154.27, 88.06) mm, rotated rx 180 ry 0 rz -180 deg; joints [-62.654, 60.281, -79.502, 63.973, 98.698, 17.207]
  Call Extruder(262.35903)
  MoveL 5999 to (239.71, 154.5, 88.06) mm, rotated rx 180 ry 0 rz 180 deg; joints [-62.708, 60.295, -79.496, 64.022, 98.673, 17.196]
  MoveL 6000 to (239.71, 154.5, 88.06) mm, rotated rx 180 ry 0 rz 180 deg; joints [-62.708, 60.295, -79.496, 64.022, 98.673, 17.196]
  Call Extruder(262.47093)
  MoveL 6001 to (239.65, 154.68, 88.06) mm, rotated rx 180 ry 0 rz 180 deg; joints [-62.754, 60.307, -79.491, 64.064, 98.652, 17.188]
  MoveL 6002 to (239.65, 154.68, 88.06) mm, rotated rx 180 ry 0 rz 180 deg; joints [-62.754, 60.307, -79.491, 64.064, 98.652, 17.188]
  Call Extruder(262.58328)
  MoveL 6003 to (239.59, 154.87, 88.06) mm, rotated rx 180 ry 0 rz 180 deg; joints [-62.801, 60.318, -79.485, 64.107, 98.631, 17.179]
  MoveL 6004 to (239.59, 154.87, 88.06) mm, rotated rx 180 ry 0 rz 180 deg; joints [-62.801, 60.318, -79.485, 64.107, 98.631, 17.179]
  Call Extruder(262.69607)
  MoveL 6005 to (239.53, 155.06, 88.06) mm, rotated rx -180 ry 0 rz 180 deg; joints [-62.847, 60.33, -79.48, 64.149, 98.61, 17.171]
  MoveL 6006 to (239.53, 155.06, 88.06) mm, rotated rx -180 ry 0 rz 180 deg; joints [-62.847, 60.33, -79.48, 64.149, 98.61, 17.171]
  Call Extruder(262.80930)
  MoveL 6007 to (239.47, 155.25, 88.06) mm, rotated rx 180 ry 0 rz 180 deg; joints [-62.893, 60.341, -79.475, 64.192, 98.589, 17.162]
  MoveL 6008 to (239.47, 155.25, 88.06) mm, rotated rx 180 ry 0 rz 180 deg; joints [-62.893, 60.341, -79.475, 64.192, 98.589, 17.162]
  Call Extruder(262.92298)
  MoveL 6009 to (239.41, 155.44, 88.06) mm, rotated rx 180 ry 0 rz -180 deg; joints [-62.939, 60.353, -79.47, 64.234, 98.568, 17.154]
  MoveL 6010 to (239.41, 155.44, 88.06) mm, rotated rx 180 ry 0 rz -180 deg; joints [-62.939, 60.353, -79.47, 64.234, 98.568, 17.154]
  Call Extruder(263.10494)
  MoveL 6011 to (239.29, 155.73, 88.06) mm, rotated rx 180 ry 0 rz 180 deg; joints [-63.018, 60.37, -79.462, 64.307, 98.534, 17.142]
  MoveL 6012 to (239.29, 155.73, 88.06) mm, rotated rx 180 ry 0 rz 180 deg; joints [-63.018, 60.37, -79.462, 64.307, 98.534, 17.142]
  Call Extruder(263.28765)
  MoveL 6013 to (239.17, 156.02, 88.06) mm, rotated rx 180 ry 0 rz 180 deg; joints [-63.097, 60.387, -79.454, 64.379, 98.5, 17.131]
  MoveL 6014 to (239.17, 156.02, 88.06) mm, rotated rx 180 ry 0 rz 180 deg; joints [-63.097, 60.387, -79.454, 64.379, 98.5, 17.131]
  Call Extruder(263.45808)
  MoveL 6015 to (239.05, 156.29, 88.06) mm, rotated rx -180 ry 0 rz 180 deg; joints [-63.17, 60.402, -79.447, 64.447, 98.469, 17.121]
  MoveL 6016 to (239.05, 156.29, 88.06) mm, rotated rx -180 ry 0 rz 180 deg; joints [-63.17, 60.402, -79.447, 64.447, 98.469, 17.121]
  Call Extruder(263.61609)
  MoveL 6017 to (238.94, 156.54, 88.06) mm, rotated rx -180 ry 0 rz 180 deg; joints [-63.238, 60.417, -79.44, 64.51, 98.44, 17.111]
  MoveL 6018 to (238.94, 156.54, 88.06) mm, rotated rx -180 ry 0 rz 180 deg; joints [-63.238, 60.417, -79.44, 64.51, 98.44, 17.111]
  Call Extruder(263.77470)
  MoveL 6019 to (238.84, 156.79, 88.06) mm, rotated rx -180 ry 0 rz 180 deg; joints [-63.306, 60.431, -79.434, 64.573, 98.411, 17.102]
  MoveL 6020 to (238.84, 156.79, 88.06) mm, rotated rx -180 ry 0 rz 180 deg; joints [-63.306, 60.431, -79.434, 64.573, 98.411, 17.102]
  Call Extruder(263.98087)
  MoveL 6021 to (238.66, 157.09, 88.06) mm, rotated rx 180 ry 0 rz -180 deg; joints [-63.401, 60.447, -79.426, 64.662, 98.373, 17.094]
  MoveL 6022 to (238.66, 157.09, 88.06) mm, rotated rx 180 ry 0 rz -180 deg; joints [-63.401, 60.447, -79.426, 64.662, 98.373, 17.094]
  Call Extruder(264.18782)
  MoveL 6023 to (238.49, 157.4, 88.06) mm, rotated rx -180 ry 0 rz 180 deg; joints [-63.497, 60.463, -79.419, 64.751, 98.335, 17.086]
  MoveL 6024 to (238.49, 157.4, 88.06) mm, rotated rx -180 ry 0 rz 180 deg; joints [-63.497, 60.463, -79.419, 64.751, 98.335, 17.086]
  Call Extruder(264.39555)
  MoveL 6025 to (238.31, 157.7, 88.06) mm, rotated rx -180 ry 0 rz -180 deg; joints [-63.592, 60.479, -79.411, 64.84, 98.297, 17.078]
  MoveL 6026 to (238.31, 157.7, 88.06) mm, rotated rx -180 ry 0 rz -180 deg; joints [-63.592, 60.479, -79.411, 64.84, 98.297, 17.078]
  Call Extruder(264.60405)
  MoveL 6027 to (238.13, 158.01, 88.06) mm, rotated rx -180 ry 0 rz 180 deg; joints [-63.687, 60.495, -79.404, 64.929, 98.259, 17.07]
  MoveL 6028 to (238.13, 158.01, 88.06) mm, rotated rx -180 ry 0 rz 180 deg; joints [-63.687, 60.495, -79.404, 64.929, 98.259, 17.07]
  Call Extruder(264.78359)
  MoveL 6029 to (237.96, 158.25, 88.06) mm, rotated rx 180 ry 0 rz -180 deg; joints [-63.774, 60.506, -79.399, 65.01, 98.227, 17.066]
  MoveL 6030 to (237.96, 158.25, 88.06) mm, rotated rx 180 ry 0 rz -180 deg; joints [-63.774, 60.506, -79.399, 65.01, 98.227, 17.066]
  Call Extruder(265.11700)
  MoveL 6031 to (237.63, 158.7, 88.06) mm, rotated rx 180 ry 0 rz 180 deg; joints [-63.934, 60.527, -79.389, 65.161, 98.166, 17.06]
  MoveL 6032 to (237.63, 158.7, 88.06) mm, rotated rx 180 ry 0 rz 180 deg; joints [-63.934, 60.527, -79.389, 65.161, 98.166, 17.06]
  Call Extruder(265.45159)
  MoveL 6033 to (237.3, 159.15, 88.06) mm, rotated rx 180 ry 0 rz 180 deg; joints [-64.094, 60.549, -79.378, 65.311, 98.106, 17.053]
  Call Extruder(266.27956)
  MoveL 6034 to (236.39, 160.19, 88.06) mm, rotated rx 180 ry 0 rz -180 deg; joints [-64.505, 60.593, -79.358, 65.7, 97.959, 17.049]
  Call Extruder(267.10747)
  MoveL 6035 to (235.35, 161.1, 88.06) mm, rotated rx -180 ry 0 rz -180 deg; joints [-64.933, 60.624, -79.343, 66.107, 97.815, 17.063]
  Call Extruder(267.27478)
  MoveL 6036 to (235.13, 161.27, 88.06) mm, rotated rx 180 ry 0 rz 180 deg; joints [-65.021, 60.628, -79.341, 66.191, 97.786, 17.069]
  MoveL 6037 to (235.13, 161.27, 88.06) mm, rotated rx 180 ry 0 rz 180 deg; joints [-65.021, 60.628, -79.341, 66.191, 97.786, 17.069]
  Call Extruder(267.60821)
  MoveL 6038 to (234.68, 161.59, 88.06) mm, rotated rx 180 ry 0 rz 180 deg; joints [-65.197, 60.637, -79.337, 66.36, 97.729, 17.079]
  MoveL 6039 to (234.68, 161.59, 88.06) mm, rotated rx 180 ry 0 rz 180 deg; joints [-65.197, 60.637, -79.337, 66.36, 97.729, 17.079]
  Call Extruder(267.94046)
  MoveL 6040 to (234.23, 161.92, 88.06) mm, rotated rx 180 ry 0 rz 180 deg; joints [-65.374, 60.646, -79.332, 66.528, 97.672, 17.09]
  MoveL 6041 to (234.23, 161.92, 88.06) mm, rotated rx 180 ry 0 rz 180 deg; joints [-65.374, 60.646, -79.332, 66.528, 97.672, 17.09]
  Call Extruder(268.05811)
  MoveL 6042 to (234.05, 162.02, 88.06) mm, rotated rx 180 ry 0 rz -180 deg; joints [-65.437, 60.648, -79.332, 66.589, 97.653, 17.096]
  MoveL 6043 to (234.05, 162.02, 88.06) mm, rotated rx 180 ry 0 rz -180 deg; joints [-65.437, 60.648, -79.332, 66.589, 97.653, 17.096]
  Call Extruder(268.26584)
  MoveL 6044 to (233.75, 162.2, 88.06) mm, rotated rx -180 ry 0 rz -180 deg; joints [-65.549, 60.65, -79.33, 66.697, 97.618, 17.107]
  MoveL 6045 to (233.75, 162.2, 88.06) mm, rotated rx -180 ry 0 rz -180 deg; joints [-65.549, 60.65, -79.33, 66.697, 97.618, 17.107]
  Call Extruder(268.47279)
  MoveL 6046 to (233.45, 162.37, 88.06) mm, rotated rx 180 ry 0 rz -180 deg; joints [-65.662, 60.653, -79.329, 66.804, 97.583, 17.117]
  MoveL 6047 to (233.45, 162.37, 88.06) mm, rotated rx 180 ry 0 rz -180 deg; joints [-65.662, 60.653, -79.329, 66.804, 97.583, 17.117]
  Call Extruder(268.67896)
  MoveL 6048 to (233.14, 162.55, 88.06) mm, rotated rx 180 ry 0 rz 180 deg; joints [-65.774, 60.656, -79.328, 66.912, 97.549, 17.128]
  MoveL 6049 to (233.14, 162.55, 88.06) mm, rotated rx 180 ry 0 rz 180 deg; joints [-65.774, 60.656, -79.328, 66.912, 97.549, 17.128]
  Call Extruder(268.86063)
  MoveL 6050 to (232.86, 162.69, 88.06) mm, rotated rx 180 ry 0 rz 180 deg; joints [-65.874, 60.657, -79.327, 67.008, 97.518, 17.138]
